(* IEC 61131-3 sources: Dev/Dev_V200/200 (part 11) *)

  	NH_M {HIDDEN} :  STRUCT 												 // m-stranka univerzalneho browsu
      // odtialto sa maze po prihlaseni
      naz         : STRING[20];                                // editovanie nazvu v hlavicke
      lvl         : USINT;                                     // level vnorenia
      lvp         : USINT;                                     // level + pg
      lng         : USINT;                                     // jazyk
      wht         : SINT;                                      // sposob ziskania dat do browsu
      iter        : SINT;                                      // iteracia
      delay       : UINT;                                      // cakanie medzi vykreslovanim (delay)
      new         : INT := -1;                                 // ND cislo pridaneho/najdeneho/vymazaneho riadka v ramci aCfg[cf]
      set         : BOOL;                                      // povolenie setup modu
      edt         : BOOL;                                      // prebieha editacia nazvu (tit)
      rgb         : BOOL;                                      // farba preRGB sa vybera aj cez slidery
      srt         : BOOL;                                      // moze preusporiadat riadky
      frm         : BOOL;                                      // aktivny vnoreny web iFrame (prekryje / deaktivuje can)
//      ref         : BOOL;                                      // prinak refreshu webu (ze prave bol refresh)
      htx         : USINT ;                                    // ktora webova stranka je zobrazena
      htt         : STRING; // := 'https://nachhouse.atlassian.net/secure/RapidBoard.jspa?rapidView=1&projectKey=NACH&selectedIssue=NACH-13' ;                             // webova adresa 'https:/www.nachhouse.sk'
      mno         : ARRAY[1..2] OF NH_OBJ_MNU;                 // zalohovanie horneho riadka pri editacii
      mnu         : ARRAY[0..3] OF NH_MNU;                    // menu
		lvd			: ARRAY[0..3] OF NH_LVL;						  // data jednotlivych vnoreni (level=lv)
      ixb         : ARRAY[0..1] OF NH_IXB;
      brw         : NH_BRW;                                   // brows
		pod			: NH_POD;
	END_STRUCT;

  	NH_WEB  {HIDDEN}:  STRUCT
		M			   : ARRAY[1.._Nh_WEB_M] OF NH_M;
      A           : ARRAY[1.._Nh_WEB_M] OF NH_CAN;
      nbr         : USINT;                         // ktory aWeb[nbr] je prave aktivny
      nrf         : USINT;								// actual count refresh display
      trg         : aTrg;
      Go          : BOOL;
	END_STRUCT;

  	NH_CAT_DSC {HIDDEN}:  STRUCT 					// categorie
 		Name        : STRING[13];
      typ         : SINT := 125;                   // filter CAT=recno(), alebo ak je > 99 tak zoznam
      dev         : USINT;                          // filter dev alebo ak je > 99 tak zoznam
      obr         : USINT := 12;
      ob0         : USINT;
      ob1         : USINT;
      Dsc         : STRING[25];

	END_STRUCT;

  	NH_STP_DSC {HIDDEN}:  STRUCT 					// categorie
 		Name        : STRING[13];
//      typ         : USINT := 255;                   // filter CAT=recno(), alebo ak je > 99 tak zoznam
      typ         : SINT := 125;                   // filter CAT=recno(), alebo ak je > 99 tak zoznam
      dev         : USINT;                          // filter dev alebo ak je > 99 tak zoznam
      obr         : USINT := 23;
	END_STRUCT;

END_TYPE

VAR_GLOBAL CONSTANT
   _e_NH_IDX_ROW        {HIDDEN}	   : NH_IDX_ROW;
	  eFilt_List			:  FILT_LIST;                                                                                      // prazdny filter
	  eFilt_List_typ		:  FILT_LIST_Typ;                                                                                      // prazdny filter

	  eRn     {HIDDEN} 	: NH_RUN_VAL2;

     eMnH     {HIDDEN} 	: NH_MNU := (     o := [(
                                        fn :=  1, wh :=  1, cm := 25  ), //       // logo
                                       (fn := 23, wh := 25, cm := 250  ),         // setup
                                       (fn :=  3, wh :=  0, cm := 20   ),         // home
                                       (fn := 41, wh := 42, cm := 21   ),         // FAV
                                       (fn := 16, wh := 17, cm := 22   ),         // rom
                                       (fn := 10, wh := 11, cm := 23   ),         // cat
                                       (fn := 27, wh := 28, cm := 24   ),         // act
                                       (fn := 49, wh :=  0, cm := 26   )]         // ON/OFF
                           );

      eMn0     {HIDDEN} : NH_MNU := (     o := [
                                       (fn :=  1, cm := 25),         // globalne nastaveia
                                       (fn := 23, cm := 250),        // setup ON/OFF
                                       (fn := 0),                    // home
                                       (fn := 41, cm :=  21),        // FAV
                                       (fn := 16, cm :=  22),        // rom
                                       (fn := 10, cm :=  23),        // cat
                                       (fn := 27, cm :=  24),        // act
                                       (fn := 0,)]);                 // ON/OFF

      eMn1     {HIDDEN} : NH_MNU := (     o := [(fn :=  0 ),  //  <
                                       (fn :=  0 ),  //  setup
                                       (fn :=  3,          cm :=  20),         // home
                                       (fn := 41,wh := 42, cm :=  21),         // FAV
                                       (fn := 16,wh := 17, cm :=  22),         // rom
                                       (fn := 10,wh := 11, cm :=  23),         // cat
                                       (fn := 27,wh := 28, cm :=  24),         // act
                                       (fn := 49,wh := 51, cm :=  26)]);       // ON/OFF

      eMvz      {HIDDEN} : NH_MNU := (     o := [(fn :=  6,wh :=   0,cm :=  31),       // <
                                       (fn :=   0,wh :=   6,cm :=   0, w:=72),  // obrazok vyssej casti
                                       (fn :=  35,wh :=  38,cm :=  33),          // 3 check
                                       (fn :=  10,wh :=  11,cm :=  34),          // 4 cat
                                       (fn :=  16,wh :=  18,cm :=  35),          // 5 all.rom / 1rom
                                       (fn := 348,wh := 348,cm :=  82),          // 6 priradit rom
//											      (fn :=  23,wh :=  24,cm :=  82),       	// 7-tune - parametre kurenia
//                                       (fn := 112,wh := 113,cm :=  36),          // visible
                                       (fn :=  39,wh :=  40,cm :=  37),          // 7-list     NESMIE SA OPRAVOVAT cm!!
                                       (fn :=  33,wh :=  34,cm :=  38)]);        // 8-play     NESMIE SA OPRAVOVAT cm!!

      eMn101     {HIDDEN} : NH_MNU := (   o := [(fn :=   6,wh :=   6,cm :=  31),          //  <
                                       (),
                                       (),
                                       (),
                                       (),
                                       (fn :=  23,wh :=  24,cm :=   3, x := xc)]);      // setup = Nastavenie parametrov

      eMn102     {HIDDEN} : NH_MNU := (   o := [(fn :=   6,wh :=   6,cm :=  31),          //  <
                                       (),
                                       (),
                                       (),
                                       (fn := 120,wh := 121,cm :=   1),          // Time
                                       (fn :=  23,wh :=  24,cm :=   3)]);        // setup = Nastavenie parametrov

      eMn103     {HIDDEN} : NH_MNU := (   o := [(fn :=   6,wh :=   6,cm :=  31),          //  <
                                       (),
                                       (fn := 122,wh := 123,cm :=   2,x:=xc-90),          // Level
                                       (fn :=  23,wh :=  24,cm :=   3,x:=xc   ),        // setup
                                       (fn :=  83,wh :=  84,cm := 121,x:=xc+90)]);           // tune predradnik / RGB

      eMn104     {HIDDEN} : NH_MNU := (   o := [(fn :=   6,wh :=   6,cm :=  31),          //  <
                                       (),
                                       (),
                                       (fn := 120,wh := 121,cm :=   1),             // Time
                                       (fn := 122,wh := 123,cm :=   2),             // Level
                                       (fn :=  23,wh :=  24,cm :=   3),             // setup
                                       (fn :=  83,wh :=  84,cm := 121)]);           // tune predradnik / RGB

      eMn105     {HIDDEN} : NH_MNU := (   o := [(fn :=   6,wh :=   6,cm :=  31),          //  <
                                       (),
                                       (fn := 120,wh := 121,cm :=   1,x:=xc-180),          // Time
                                       (fn := 122,wh := 123,cm :=   2,x := xc-90),          // Level + Ramp ON/OFF
                                       (fn := 124,wh := 125,cm :=   4,x := xc),          // COLOR
                                       (fn :=  23,wh :=  24,cm :=   3,x := xc+90),          // setup = Nastavenie parametrov
                                       (fn :=  83,wh :=  84,cm := 121,x := xc+180)]);        // tune predradnik / RGB

      eMnTLA   {HIDDEN} : NH_MNU := (   o := [(fn :=   6,wh :=   6,cm :=  31),          //  <
                                       (),
                                       (fn :=  33,wh :=  34,cm :=   5,x := 205),          // PLAY = priradenie
                                       (fn :=  23,wh :=  24,cm :=   6,x := 385)]);        // setup

      eMnWSB   {HIDDEN} : NH_MNU := (   o := [(fn :=   6,wh :=   6,cm :=  31),          //  <
                                       (),
                                       (fn :=  33,wh :=  34,cm :=   5,x := 205),          // PLAY = priradenie
                                       (fn := 204,wh := 205,cm := 120,x := 295),          // LED WSB
                                       (fn :=  23,wh :=  24,cm :=   6,x := 385)]);        // setup

      eMnPIR     {HIDDEN} : NH_MNU := (   o := [(fn :=   6,wh :=   6,cm :=  31),          //  <
                                       (fn :=   0,wh :=   0,cm :=   0),
                                       (fn :=   0,wh :=   0,cm :=   0),
                                       (fn := 215,wh := 216,cm :=  10,x := 115),          // Day
                                       (fn := 217,wh := 218,cm :=  10,x := 205),          // Evening
                                       (fn := 219,wh := 220,cm :=  10,x := 295),          // Night
                                       (fn := 221,wh := 222,cm :=  10,x := 385),          // Morning
                                       (fn :=  23,wh :=  24,cm :=   9,x := 475)]);        // setup = Nastavenie parametrov

      eMnUsr     {HIDDEN} : NH_MNU := (   o :=
                                      [(fn :=   6,wh :=   6,cm :=  31),          //  <
                                       (fn :=  32,wh :=  25,cm := 101),          //  +
                                       (fn :=   0,wh :=   0,cm :=   0),
                                       (fn :=   0,wh :=   0,cm :=   0),
                                       (fn :=  79,wh :=  79,cm :=  55),          // Users
                                       (fn := 285,wh := 286,cm :=  56),          // Web
                                       (fn :=   0,wh :=   0,cm :=   0),
                                       (fn :=   0,wh :=   0,cm :=   0)]);

(*
   _NhObrXYZ {HIDDEN} :  ARRAY [-10..-1,0..3] OF INT :=                 // obrazky podla nejakej podmieny (typ,stav...)
            [
//                21, 79,315, 21,             // -11 ZONE
               258, 82,  0,  0,             // -10 RH,CO2,CO
               508,216,166,507,             // -9 BRA  garaz,brana,branicka,zavora
               168,169,169,168,             // -8 SIR/STROB/
               183,184,185,186,             // -7 HET
                60, 60, 60, 60,             // -6  FAV dash/quick/FAV all/FAV user
                17, 19, 15,17,              // -5  ROM   In/OUT/pivnica
               106,107,  0,  0,             // -4  TLA   1/2
               102,103,104,105,             // -3  WSB   2/4/8/5
               100, 99,100,100,             // -2  termoventil : TVE, spirala
               161,162,  0,  0              // -1  teploty  :    miestnost,vonku //,podlaha,kotol

            ];

   // wht   :  index _NhStavDev[wht] odkial sa zoberi parametre do prikazu pre zobrazenie
   //          _NhVal2(wh := _NhStaDev[s].wht, obr := _NhStaDev[s].val);
   //             wh    - je bud podklad, alebo jednorazova prikaz, ktory nadefinuje vykreslenie
   //             obr   - ak si ho funkcia (wh) inak nespracuje, tak je to obrazok
   // val   :  ak je > 0 = cislo obrazka
   //          ak je < 0 je to odkaz na _NhObrXYZ[val], kde su obrazky podla nejakeho kriteria k DEV (vacsinou xCfg^.typ). rozduje funkcia _NhObrNbr()

   _NhObrDev  :  ARRAY [0.._Nh_CFG] OF NH_DEF_OBR :=     // definicia zakladnych obrazkov a obrazkov stavu (stav=odkaz) pre  DEV
            [
            (wht :=   0, val :=  23),      //  wht = index _NhStavDev[wht], val = cislo obrazka   ak je val < 0 potom je odkaz na _NhObrXYZ[val]
            (wht :=   1, val :=  -5),      //  1 ROM INR/EXT
            (wht :=   0, val :=  11),      //  2 CAT
            (wht :=   0, val :=  21),      //  3 ZON  stavovy obrazok sa definuje v _NhBrw6 CASE:9, hlavny obrazok:=21
            (wht :=  27, val :=  30),      //  4 SCN
            (wht :=  25, val :=  28),      //  5 ACT  0/34

//            (wht :=  29, val :=  -7),      //  6 HET
            (wht :=   0, val := 183),      //  6 HET
            (wht :=  42, val :=  95),      //  7 KOT
            (wht :=  42, val := 100),      //  8 TVE
            (wht :=   0, val := 101),      //  9 CER

            (wht :=   5, val :=  62),      // 10 SVD
            (wht :=   7, val :=  63),      // 11 SVA
            (wht :=   9, val :=  64),      // 12 RGB

            (wht :=   0, val :=  -3),      // 13 WSB     stavovy obrazok sa definuje v _NhBrw6
            (wht :=   0, val :=  -4),      // 14 TLA     stavovy obrazok sa definuje v _NhBrw6
            (wht :=  23, val :=  87),      // 15 PIR
            (wht :=   3, val :=  -1),      // 16 TER
            (wht :=   3, val := 163),      // 17 TEH
            (wht :=   3, val := 164),      // 18 TEK
            (wht :=   4, val :=  86),      // 19 LUX
            (wht :=   0, val :=  -6),      // 20 FAV
            (wht :=  11, val :=  73),      // 21 ZAS
            (wht :=   0, val :=  78),      // 22 USR
            (wht :=  30, val :=  70),      // 23 VENT
            (wht :=   0, val :=  97),      // 24 KEY
            (wht :=   0, val := 298),      // 25 SMART-WAY
            (wht :=   0, val :=   1),      // 26   POI
            (wht :=   0, val :=   1),      // 27 H2O
            (wht :=   0, val :=   1),      // 28 FIR
            (wht :=   0, val :=   1),      // 29 GAS
            (wht :=   0, val := 110),      // 30 MAR
            (wht :=  44, val := 114),      // 31 ROL
            (wht :=  30, val :=  -8),      // 32 SIR
            (wht :=  35, val :=  91),      // 33 DOR
            (wht :=  33, val :=  92),      // 34 WIN
            (wht :=   0, val := 197),      // 35 BLI
            (wht :=   0, val :=   1),      // 36   XXX
            (wht :=  50, val :=  -9),      // 37 BRA
            (wht :=   0, val :=   1),      // 38 RFI-snimace
            (wht :=   0, val :=   1),      // 39 RFK-karty
            (wht :=   0, val := 310),      // 40 TGL
            (wht :=   0, val := -10),      // 41 COX  (RH,CO2,CO)
            (wht :=   0, val := 290),      // 42 DALI-M
            (wht :=   0, val := 063),      // 43 DALI-S
            (wht :=   0, val := 029)       // 44 DALI-G
            ];

   // _NhStaDev: vykreslenie obraka podlastavu DEV vo funkcii : _NhVal2(wh := _NhStaDev[].wht, obr := _NhStaDev[].val);
   // jedno dev v _NhStaDev ma viac viet, podla stavu
   //    _NhStaDev[wht+0]  := 1.veta ked xDev^.ou.val = 0.0;
   //    _NhStaDev[wht+1]  := 2.veta ked xDev^.ou.val > 0.0;
   //    _NhStaDev[wht+2]  := 3.veta ked moze existovat ine kriterium unikatne k DEV

   // vsetko sa vyrobi v _NhShwObj() ked xO^.wh := 3

   _NhStaDev {HIDDEN} :  ARRAY [0.._Nh_CFG] OF NH_DEF_OBR :=               // zobrazenie stavy DEV (obrazky, hodnoty, ikony ,,,)
            [
            (wht :=   0, val :=  23),      //  0 nic (obrazok setup)
            (wht :=   1, val :=   0),        //  1 ROM - zobrazenie teploty
            (),                              // 2 - volne
//            (wht :=  18, val :=  66),        //  2 ZON - zobrazenie teploty
            (wht :=   1, val :=   0),        //  3 teplota miestnosti,vonku,podlahy,kotla... podla typ
            (wht :=   2, val :=   0),        //  4 LUX - zobrazenie osvetlenia
            (wht :=  10, val :=  -1),        //  5 SVD - OFF   (-1 znamena ze sa nevykresli ziadny obrazok !!!)
//            (wht :=  11, val :=   0),        //  6 SVD - ON - v zltom kruhu s gradientom
            (wht :=  17, val := 201),        //  6 SVD - ON - v zltom kruhu s gradientom
            (wht :=  10, val :=  -1),        //  7 SVA - OFF
//            (wht :=  12, val :=   0),        //  8 SVA - lvl v zltom kruhu s gradientom
            (wht :=  17, val := 201),        //  8 SVA - ON - v zltom kruhu s gradientom
            (wht :=  10, val :=  -1),        //  9 RGB - OFF
//            (wht :=  12, val :=   0),        // 10 RGB - lvl v zltom kruhu s gradientom
            (wht :=  17, val := 201),        // 10 RGB - ON - v zltom kruhu s gradientom

            (wht :=  18, val :=  73),       // 11 ZAS - NEURCENY-OFF            sivy + obrazok
            (wht :=  18, val :=  62),       // 12 ZAS - SVE-OFF                 sivy + obrazok
            (wht :=  18, val :=  50),       // 13 ZAS - STYKAC-OFF               sivy + obrazok
            (wht :=  18, val :=  61),       // 14 ZAS - HET-OFF                 sivy + obrazok
            (wht :=  18, val := 159),       // 15 ZAS - NABIJ.STANICA-OFF        sivy + obrazok
            (wht :=  18, val :=  73),       // 16 ZAS - rezerva-OFF              sivy + obrazok

            (wht :=  13, val := 202),       // 17 ZAS - NEURCENY-ON             zeleny + obrazok
            (wht :=  17, val := 201),       // 18 ZAS - SVD-ON                  zlty   + obrazok
            (wht :=  13, val := 213),       // 19 ZAS - SYKAC ON                 zeleny + obrazok
            (wht :=  13, val := 203),       // 20 ZAS - HET-ON                  zeleny + obrazok
            (wht :=  13, val := 214),       // 21 ZAS - NABIJACIA STANICA-ON    zeleny + obrazok
            (wht :=  13, val := 202),       // 22 ZAS - rezerva -ON             zeleny + obrazok

            (wht :=  10, val :=  -1),       // 23 PIR - pir je v klude, neodpocitava sa nic
            (wht :=  16, val :=  89),       // 24 PIR - prihadza signal          cierna postava v modrom

            (wht :=  18, val :=  28),       // 25 ACT - OFF sipka v sivom kruhu
            (wht :=  20, val :=  28),       // 26 ACT - ON sipka v Azurovom kruhu bez gradientu

            (wht :=  18, val :=  30),       // 27 SCN - OFF scn v sivom kruhu
            (wht :=  14, val := 207),       // 28 SCN - ON  scn v oranzovom kruhu

            (wht :=   1, val :=   0),       // 29 HET - zobrazenie teploty

            (wht :=  10, val :=  -1),       // 30 VEN - OFF
            (wht :=  13, val := 215),       // 31 VEN - ON - v modrom kruhu s gradientom

            (wht :=   4, val :=   0),       // 32 TVE - vystredene cislo v azurovom kruhu

            (wht :=  18, val :=  -1),       // 33 WIN - OFF
            (wht :=  14, val :=  92),       // 34 WIN - ON - v modrom kruhu s gradientom

            (wht :=  18, val :=  -1),       // 35 DOR - OFF
            (wht :=  14, val :=  91),       // 36 DOR - ON - v modrom kruhu s gradientom

            (wht :=  18, val :=  66),       // 37 ZON - Unlocked 0
            (wht :=  14, val :=  67),       // 38 ZON - Lock   1/2
            (wht :=  15, val :=  67),       // 39 ZON - Lock full
            (wht :=  18, val :=  66),       // 40 ZON - Locking
            (wht :=  18, val :=  66),       // 41 ZON - Unlocking

            (wht :=  10, val :=  -1),       // 42 TVE - OFF
            (wht :=  40, val :=   0),       // 43 TVE - cerveny kruh s cislo v strede

            (wht :=  18, val := 114),       // 44 ROL - OFF  0%      dn - zatiahnute     sivy
            (wht :=  14, val := 115),       // 45 ROL - viac 1-99%   up/dn - povytiahnute      oranzovy
            (wht :=  23, val := 117),       // 46 ROL - pohyb hore               cerveny
            (wht :=  23, val := 118),       // 47 ROL - pohyb dolu               cerveny
            (wht :=  90, val := 501),       // 48 ŽAL - zatienene    siva
            (wht :=  90, val := 500),       // 49 ŽAL - zodtienene   biela

            (wht :=  18, val := 509),       // 50 GAR - OFF  0%         sivy
            (wht :=  23, val := 510),       // 52 GAR - otvorene  100%  cerveny
            (wht :=  18, val := 216),       // 53 BRANA - OFF  0%         sivy
            (wht :=  15, val := 217),       // 54 BRANA - otvorene  100%  cerveny gradient
            (wht :=  18, val := 166),       // 55 BRANICKA - OFF  0%         sivy
            (wht :=  23, val := 167),       // 56 BRANICKA - otvorene  100%  cerveny
            (wht :=  21, val := 506),       // 55 BRANICKA - OFF  0%         sivy
            (wht :=  23, val := 507)        // 56 BRANICKA - otvorene  100%  cerveny

         ];

   // tito parametre sa posielaju do _NhVal2(wh := _NhStaCat[s].wht, obr := _NhStaCat[s].val);
   // wht : funkcia
   // val : obrazok
   // vsetko sa vyrobi v _NhShwObj() ked xO^.wh := 2
*)

END_VAR

VAR_GLOBAL CONSTANT

	{ $ IF _nh_Cust = 0 OR _Nh_CUST = 1} 	 // vsetko

      _ePg0   : NH_PG_HOME :=
      (
      Hom := ( ob := [
               ( wh:= 1, x := xc,     y := yyc- 30,  w := 180,  fn := 255 ),                                  // domcek
               ( wh:= 1, x := xc,     y := yyc- 55,  w :=  32,  fn := 0 ),                                   // day/night vnutri
               ( wh:= 0, x := xc+ 40, y := yyc-120,  w :=  32,  fn := 140 ),                                  // day/night vonku
               ( wh:= 1, x := xc,     y := yyc-  5,  w :=  80,  fn :=  92,   cm := 50,    cf := (c:=2, n:=17)),   // okno
               (),
//               ( x := xc+ 30, y := yc+ 90,  w :=  50,  wh := 0,  fn :=  92, h := -70, FgC := 1, BgC := 8,   cf := (c:=2, n:=18)),   // otvorene dvere ( h > 0 : vymaze aj kruh pod obrazkom)
               ( x := xc- 30, y := yyc+ 90,  w :=  50,  wh := 0,  fn := 111, h := -70, FgC := 8, BgC := 1,   cf := (c:=2, n:=23)),   // otvoreny garaz
               ( x := xc+100, y := yyc+ 20,  w :=  50,  wh := 0,  fn :=  77, h :=   0,                       cf := (c:=2, n:=24)),  // otvorena brana/branicka
               ( x := xc- 45, y := yyc-130,  w :=  75,  wh := 1,  fn := 132, h :=   0,                       cf := (c:=2, n:=11)),  // fotovoltaika

               ( wh:=4, x := xc-60, y := yyc+45, w:=58, h:=48, fn := 0, FgC := 0, BgC := 0,   cf := (c:=1, n:=1)),   // otvorene dvere ( h > 0 : vymaze aj kruh pod obrazkom)
               ( wh:=4, x := xc-60, y := yyc+45, w:=58, h:=48, fn := 91, cm := 50,   cf := (c:=2, n:=18)),   // otvorene dvere ( h > 0 : vymaze aj kruh pod obrazkom)
               (BgC := 13)
                     ]),

      dsh :=  ( ob := [

               (x := 0,      y:= 0, wh := 0),
               (x := xc,     y:= yyc-253, w := 130, wh := 2, cm:=50),   // 1.kruznica pod obr.1 prvy hore
               (x := xc+158, y:= yyc-183, w := 130, wh := 2, cm:=50),   // 2.kruznica pod obr.2
               (x := xc+210, y:= yyc- 25, w := 130, wh := 2, cm:=50),   // kruznica pod obr.3 - vprav v strede
               (x := xc+158, y:= yyc+133, w := 130, wh := 2, cm:=50),   // kruznica pod obr.4
               (x := xc,     y:= yyc+203, w := 130, wh := 2, cm:=50),   // kruznica pod obr.5 - dolu
               (x := xc-158, y:= yyc+133, w := 130, wh := 2, cm:=50),   // kruznica pod obr.6
               (x := xc-210, y:= yyc- 25, w := 130, wh := 2, cm:=50),   // kruznica pod obr.7 - vlavo v strede
               (x := xc-158, y:= yyc-183, w := 130, wh := 2, cm:=50)    // kruznica pod obr.8
                     ]),

      Qck :=  ( ob := [

               (x := xc-220, y := yy2-70, w := 64, wh := 0),                      // 1 - preve zprava
               (x := xc-220, y := yy2-65, w := 64, wh := 2, cm:=50),                      // 1 - preve zprava
               (x := xc-130, y := yy2-65, w := 64, wh := 2, cm:=50),
               (x := xc- 40, y := yy2-65, w := 64, wh := 2, cm:=50),
               (x := xc+ 50, y := yy2-65, w := 64, wh := 2, cm:=50),
               (x := xc+140, y := yy2-65, w := 64, wh := 2, cm:=50),
               (x := xc+230, y := yy2-65, w := 64, wh := 2, cm:=50),                      // 6 - posledne zlava
               (x := xc+320, y := yy2-65, w := 64, wh := 2, cm:=50),                      // 7 - dalej
               ()
                     ]),
      xy := [
               (),
               (x := 380, y := 275),
               (x := 490, y := 400),
               (x := 490, y := 562),
               (x := 380, y := 693),
               (x := 205, y := 693),
               (x :=  87, y := 569),
               (x :=  87, y := 400),
               (x := 200, y := 275)
               ],

      );

	{ $ END_IF }

	{ $ IF _Nh_CUST = 2} 	                // Futbal.stadion HE
      _ePg0 : NH_PG_HOME :=
      (
      Home := ( ob := [
               ( x := xc,    y:= yc- 20, w:= 600, wh:=1,          fn := 300 ),                    // futb.stadion
//               ( x := xc+15, y:= yc- 20, w:= 160, wh:=1,          fn := 301 ),                    // futb.stadion
               ()
                     ]),
      Dash :=  ( ob := [
               (x := xc-200, y:= yc+220, w := 110, wh := 2 , cf := (c := 2)),   // kruznica pod obr.1 prvy hore
               (x := xc-200, y:= yc+ 65, w := 110, wh := 2 , cf := (c := 2)),   // kruznica pod obr.2
               (x := xc-200, y:= yc-105, w := 110, wh := 2 , cf := (c := 2)),   // kruznica pod obr.3 - vprav v strede
               (x := xc-200, y:= yc-260, w := 110, wh := 2 , cf := (c := 2)),   // kruznica pod obr.4
               (x := xc+195, y:= yc-260, w := 110, wh := 2 , cf := (c := 2)),   // kruznica pod obr.5 - dolu
               (x := xc+195, y:= yc-105, w := 110, wh := 2 , cf := (c := 2)),   // kruznica pod obr.6
               (x := xc+195, y:= yc+ 65, w := 110, wh := 2 , cf := (c := 2)),   // kruznica pod obr.7 - vlavo v strede
               (x := xc+195, y:= yc+220, w := 110, wh := 2 , cf := (c := 2))    // kruznica pod obr.8
                     ]),

      Quick :=  ( ob := [

               (x := xc+320, y := y2-60, w := 64, wh := 2),
               (x := xc+230, y := y2-60, w := 64, wh := 2),
               (x := xc+140, y := y2-60, w := 64, wh := 2),
               (x := xc+ 50, y := y2-60, w := 64, wh := 2),
               (x := xc- 40, y := y2-60, w := 64, wh := 2),
               (x := xc-130, y := y2-60, w := 64, wh := 2),
               (x := xc-220, y := y2-60, w := 64, wh := 2),
               (x := xc-310, y := y2-60, w := 64, wh := 2),
               (),
               (w := 48, wh := 100)                    // weather
                     ]),

      );

      eMnHfs     : NH_MNU := (  n := 3,                                               // len obrazok HOME
                              o := [(fn :=  1),(fn := 0),
                                       (wh := 4, fn := 4, cm :=20, x:=xc, y:= y2+55),         // home
                                       (wh := 0, fn := 0, cm :=0 ),
                                       (wh := 0, fn := 0, cm :=0 ),
                                       (wh := 0, fn := 0, cm :=0 ),
                                       (wh := 0, fn := 0, cm :=0 ),
                                       (wh := 0, fn := 0, cm :=0 )
                                       ]);

   { $ END_IF }

	{ $ IF _Nh_CUST = 3} 	                // zimny stadion HE
      _ePgHome : NH_PG_HOME;
	{ $ END_IF }
END_VAR

//      pHet     : ARRAY[0..1,1..4] OF USINT := [170,172,174,176, 171,173,175,177];                                       // HeatMode */1/2/3/ manual/program
//      pTve     : ARRAY[0..1,0..3] OF USINT := [ 49,172,174,176,  52,173,175,177];                                       // Tve    Off/1/2/3/ manual/program

VAR_GLOBAL CONSTANT

(*
   // [OFF/ON, HET/TVE, A/1/2/3]      HET, TVE  OFF..ON    A,0,1,2,3              [0,OFF,            n] [0,ON,             n]
   _ObrHetPVP     {HIDDEN}   : ARRAY[ 0  ..  2, 0..   1,   0 ..    4] OF USINT := [222,170,172,174,176,  223,171,173,175,177, // HET: [0,OFF/ON, PRG/0/1/2/3/4 ]
                                                                                   222, 54,172,174,176,  223,193,173,175,177, // VEN: [1,OFF/ON, PRG/0/1/2/3/4 ]
                                                                                   220, 54,172,174,176,  221,193,173,175,177  // TVE: [2,OFF/ON, MAN/0/1/2/3/4 ]
*)

   _NhListObr     {HIDDEN}   : NH_LIST_OBR;
   _NhTypeMnu     {HIDDEN}   : NH_TYPE_MNU;
	_NhDsh			{HIDDEN}   : NH_DSH;
   _eRowHed       {HIDDEN}	  : NH_ROW_H;                   // cisla hlavicka riadka
   _eSld          {HIDDEN}	  : NH_SLD_DAT;
   _eFil          {HIDDEN}	  : NH_FIL;
   _eWht          {HIDDEN}   : NH_TCH_WHT;
   _eTch          {HIDDEN}	  : NH_TCH;                     // prazdny touch
   _eRowH         {HIDDEN}	  : NH_ROW_H;                    // prazdna hlavicka riadka
//   _ObjDay        {HIDDEN}   : NH_POI_DAY_XY;
   _NhObrLeds     {HIDDEN}   : ARRAY[1..4] OF USINT := [210,209,212,208];    // R,G,B,SH

//	_NhObjCfgBlk    :  NH_OBJ_DAT  :=          // PIR
//      (wh:= 0, x:=125,  y:=109,  w:=48, h:= 68, FgC:=4,  BgC:=2,  fn:=0            ); // 5 Blk
	_NhObjD1pir    :  NH_OBJ_DAT  :=          // PIR
      (wh:= 0, x:=125,  y:=109,  w:=50, h:=68 , FgC:=7,  BgC:=2,  fn:=0, cf:=(c:=5)); // 6 PIR day mde

END_VAR

VAR_GLOBAL
	aWeb			      : NH_WEB;

   yRn         {HIDDEN}     : NH_RUN_VAL2;

   xM          {HIDDEN}     : PTR_TO NH_M;
   xA          {HIDDEN}     : PTR_TO NH_CAN;
   xB          {HIDDEN}     : PTR_TO NH_BRW;
   xL		      {HIDDEN}     : PTR_TO NH_LVL;
   xF		      {HIDDEN}     : PTR_TO NH_FIL;
   xU          {HIDDEN}     : PTR_TO NH_MNU;
   xR          {HIDDEN}     : PTR_TO NH_ROW;
   xR2         {HIDDEN}     : PTR_TO NH_ROW;
   xRowO			{HIDDEN}     : PTR_TO NH_ROW_O;
	xS          {HIDDEN}     : PTR_TO NH_SLD_DAT;
   xO          {HIDDEN}     : PTR_TO NH_OBJ_DAT;
   xO2         {HIDDEN}     : PTR_TO NH_OBJ_DAT;
   xOh         {HIDDEN}     : PTR_TO NH_OBJ_123;
   xOh2        {HIDDEN}     : PTR_TO NH_OBJ_123;

   x4o         {HIDDEN}     : PTR_TO NH_OBJ_4O1;
	xRo 			{HIDDEN}		 : PTR_TO NH_OBJ_ROL;
//	yRo 			{HIDDEN}	AT aWeb.M[1].brw.r[14]	: NH_OBJ_ROL;
	yRo 			{HIDDEN}		:  NH_OBJ_ROL;
	x124			{HIDDEN}		:  PTR_TO NH_OBJ_124;
	y124			{HIDDEN}		:  NH_OBJ_124;

   xoDsh       {HIDDEN}     : PTR_TO NH_OBJ_DSH;

   xOm         {HIDDEN}     : PTR_TO NH_OBJ_MNU;
   xIxB        {HIDDEN}	    : PTR_TO NH_IXB;
   xIdx        {HIDDEN}	    : PTR_TO NH_IDX;
 	yIdxR			{HIDDEN}	    : NH_IDX_ROW;

   ky2          {HIDDEN} : INT := 915;                    // koniec browsu = zaciatok spodneho menu
   kyr          {HIDDEN} : INT := 132;                    // vyska riadku
   kyc          {HIDDEN} : INT := 510;                    // stred Y
   kyb          {HIDDEN} : INT := 800;                    // celkova vyska browsu
   yk           {HIDDEN}       : REAL;
   yLVL                   : NH_LVL;
   aAcc                             : NH_WEB_ACC;                      // riadiaca premenne
   CustomizedLoginPage AT %S355.1    {HIDDEN}   : BOOL := true;                     // povolenie Cust pristupu (prekopirovat XML do web/import)
   targetPage                        {HIDDEN} : STRING[20] := '001_NHM.XML';           // nazov stranky na ktoru presmeruje REDIR.XML
   aHtt                              {HIDDEN} : STRING[80] ; //:= '_NH_USR_.XML';
//   pageLogout                       : ARRAY [1..3] OF STRING[20];       //

END_VAR

VAR_GLOBAL		// docasne pomocne premenne
   yS          				{HIDDEN}     : NH_SLD_DAT;
   y4o         				{HIDDEN}     : NH_OBJ_4O1;
   yOh         				{HIDDEN}     : NH_OBJ_123;
	yoDsh       				{HIDDEN}     : NH_OBJ_DSH;
	_NhObjO4rom 				{HIDDEN}     :  NH_OBJ_4O1;
	_NhObjO4sta 				{HIDDEN}     :  NH_OBJ_4O2;
   xCan        				{HIDDEN}     : PTR_TO TCanvasData;
END_VAR

FUNCTION _NhVal2  : BOOL           // nadefinovanie stavoveho obrazka/textu pre kategoriu
   VAR_INPUT
      xy       : BOOL;                    // znamena, ze sa text vypisuje len pre to co je v x,y, inak pre xO^.x + x
      noxy     : BOOL;                    // text sa vypise od nastavenej pozicie
      nofmt    : BOOL;                    // text sa neformatuje
      crc      : BOOL;                    // vykresluje sa kruh
      box      : BOOL;                    // vykresluje sa obdlznik
      fil      : BOOL := true;            // vykresluje sa obsah kruhu/obdlznika
   	wrk		: BOOL;
	   wh       : USINT;                   // predvolba
      grd      : USINT;                   // typ gradientu
      obr      : INT;                     // vykresli sa obrazok
      txt      : SINT   := -1;            // vypise sa text (-1 := nic sa nevypise)
		nTxt		: INT;							// cislo textu
      FgC      : USINT  := 2;             // GCOLOR_LTGRAY;
      BgC      : USINT  := 1;             // GCOLOR_BLACK;
      FgT      : USINT  := 4;             // GCOLOR_WHILE;
      fmt      : INT    := 2;             // formatovanie textu (stred riadka, stred textu)
      wC       : INT    ;                 // priemer kruhu/sirka boxu
      hB       : INT    ;                 // vyska boxu
      wO       : INT    ;                 // velkost obrazka
      wT       : INT := 22   ;            // velkost textu
      wL       : USINT  := 2;             // hrubka kruznice / oramovanie kruhu
      x,y      : INT;                     // korekcie
      r        : INT    := 2;             // polomer Rounbow
      ob       : SINT := -1;               // namapuje xO
      val      : STRING[10];              // nieco naforpatovane pre zobrazenie ako text
   END_VAR
   VAR_TEMP
      n        : INT;
   END_VAR
   _NhVal2 := true;
   IF ob > -1 THEN
      xO := ADR(xR^.o.ob[ ob ]);
   END_IF;

   IF wC = 0 THEN
      wC := xO^.w;
   END_IF;
   IF wO = 0 THEN
//      wO := wC-7;
      wO := wC/5*4;
   END_IF;
   IF hB = 0 THEN
      hB := wC;
   END_IF;
   IF wT = 0 THEN
      wT := xO^.h;
   END_IF;
   CASE wh OF                                                          // jednoucelovo nadefinovane predvolby

      0: //bez predvolby = vypisuje sa podla toho co prislo v parametroch ( crc,obr,txt....)
         ;

    100: // normalna teplota z al.ou.val, formatovanie textu podla xO^.fn    , vyska xO^.h, farba podla FgC
         FgT := xO^.FgC; txt := 10; wT := xO^.h; fmt := xO^.fn; fil := false;
    101: // % (luxy,CO) z al.ou.val, formatovanie textu podla xO^.fn, vyska xO^.h
         FgT := xO^.FgC; txt := 11; wT := xO^.h; fmt := xO^.fn; fil := false;
    102: // oranzovy gradient-kruh s ciernym 'ON'
         fil :=1; crc := 1; grd := 11;  FgC :=15; BgC :=  4; FgT := 1; txt := 2; wT := 18;
    103: // azurovy gradient-kruh s ciernym 'ON'
         fil :=1; crc := 1; grd := 11;  FgC :=3; BgC :=  4; FgT := 1; txt := 2; wT := 18;

    109: // modry gradient-kruh s cislom v strede z al.ou.val
         fil :=1; crc := 1; grd := 11;  FgC := 3; BgC :=  3; FgT := 4; txt :=15; wT := 22; fmt := 2;
    110: // zlty gradient-kruh s cislom v strede z al.ou.val
         fil :=1; crc := 1; grd := 11;  FgC := 5; BgC :=  4; FgT := 1; txt :=15; wT := 22; fmt := 2;
    111: // Zeleny gradient-kruh s cislom v strede z al.ou.val
         fil :=1; crc := 1; grd := 11;  FgC := 8; BgC :=  4; FgT := 1; txt :=15; wT := 22; fmt := 2;
    112: // Oranzovy gradient-kruh s cislom v strede z al.ou.val
         fil :=1; crc := 1; grd := 11;  FgC :=15; BgC :=  4; FgT := 1; txt :=15; wT := 22; fmt := 2;
    113: // Azurovy  gradient-kruh s cislom v strede z al.ou.val
         fil :=1; crc := 1; grd := 11;  FgC := 3; BgC :=  4; FgT := 1; txt :=15; wT := 22; fmt := 2;
    114: // Purpurovy gradient-kruh s cislom v strede z al.ou.val
         fil :=1; crc := 1; grd := 11;  FgC := 28; BgC := 2; FgT := 4; txt :=15; wT := 22; fmt := 2;
    115: // Cerveny gradient-kruh s cislom v strede z al.ou.val
         fil :=1; crc := 1; grd := 11;  FgC := 7; BgC :=  4; FgT := 1; txt :=15; wT := 22; fmt := 2;
    116: // Biely gradient-kruh s cislom v strede z al.ou.val
         fil :=1; crc := 1; grd := 11;  FgC := 4; BgC :=  2; FgT := 1; txt :=15; wT := 22; fmt := 2;
    117: // Zeleny kruh bez grd s cislom z VR cierny text - pre CHECK/analog
	      fil :=1; crc := 1; grd := 1;  FgC := 8; BgC :=  8; FgT := 1; txt := 3; wT := 22; fmt := 2;
    118: // Zeleny kruh bez grd s cislom z VR cierny text - pre CHECK/DIGITAL
	      fil :=1; crc := 1; grd := 1;  FgC := 8; BgC :=  8; FgT := 1; txt := 2; wT := 22; fmt := 2;
    120: // silne sve tlo-cerveny  kruh + gradient
         fil :=1; crc := 1; grd := 11;  FgC := 18; BgC :=  4;   //BgC :=  4;

    150: // Cerveny gradient-kruh s cislom v strede z al.ou.sta
         fil :=1; crc := 1; grd := 11;  FgC := 7; BgC :=  4; FgT := 1; txt :=16; wT := 22; fmt := 2;
    151: // Cerveny gradient-kruh s cislom v strede z al.ou.ex
         fil :=1; crc := 1; grd := 11;  FgC := 7; BgC :=  4; FgT := 1; txt :=17; wT := 22; fmt := 2;

    160: // tmavo-cerveny kruh + svetly gradient
         fil :=1; crc := 1; grd := 11;  FgC :=28; BgC :=  4;
    161: // purpurovy kruh + tmavy gradient
         fil :=1; crc := 1; grd := 13;  FgC :=28; BgC :=  1;   //BgC :=  4;

    170: // tmavo-modry obdlznik bez gradientu
         fil :=1; box := 1; grd := 1;   FgC :=4; BgC :=  9;
    171: // svetlo-modry obdlznik bez gradientu
         fil :=1; box := 1; grd := 11;  FgC :=4; BgC := 22;   //BgC :=  4;

      1: // teplota v browse
         FgT := xO^.FgC; txt := 10; wT := 32; fmt := 1; x := 30; y := -5;    // skoriguje suradnice vypisu teploty - posunie do prava a odtial sa vykresluje do lava
//         FgT := xO^.FgC; txt := 10; wT := xO^.h; fmt := 1; x := 30; y := -5;    // skoriguje suradnice vypisu teploty - posunie do prava a odtial sa vykresluje do lava
      2: // % osvetlenia v browse
         FgT := xO^.FgC; txt := 11; wT := 28; fmt := 1; x := 30; y := -5;
      3: // lx v browse
         FgT := xO^.FgC; txt := 12; wT := 28; fmt := 1; x := 30; y := -5;
      4: // vystredene cislo v sivom kruhu s gradientom
         FgT := 4; txt := 3; wT := 20; fmt := 2;               // cislo bielou
         crc := 1; grd := 11;  FgC := 2; BgC :=  1; wC := 60;

      9: // kruh bez gradientu vypln farbou Bgc, bez oramovanie pripadny text farbou FgC, text podla poslanych parametrov
         fil :=1; crc := 1; grd := 2; Fgc:= BgC; FgT := 1; wL := 0;

//         fil :=1; crc := 1; grd := 2;  FgC := 8; BgC :=  8; FgT := 1;

     10: // sivy gradient-kruh s bielym 'OFF'
         fil :=1; crc := 1; grd := 11;  FgC := 2; BgC :=  1; FgT := 4; txt := 1; wT := 19;

     11: // zlty gradient-kruh s ciernym 'ON'
         fil :=1; crc := 1; grd := 11;  FgC := 5; BgC :=  4; FgT := 1; txt := 2; wT := 18;

     12: // zlty gradient-kruh s cislom v strede
         fil :=1; crc := 1; grd := 11;  FgC := 5; BgC :=  4; FgT := 1; txt := 3; wT := 22;

     13: // zeleny   kruh + gradient
         fil :=1; crc := 1; grd := 11;  FgC := 8; BgC :=  4;
     14: // oranzovy kruh + gradient
         fil :=1; crc := 1; grd := 11; FgC := 15; BgC :=  4; //FgC := 6; BgC :=  4;
         IF obr > 0 THEN
            wO := wC/4*3;
         END_IF;
     15: // sve tlo-cerveny  kruh + gradient
         fil :=1; crc := 1; grd := 11;  FgC := 7; BgC :=  4;   //BgC :=  4;
     16: // azurovy  kruh + gradient
         fil :=1; crc := 1; grd := 11;  FgC := 3; BgC :=  4;
     17: // zlty gradient-kruh
         fil :=1; crc := 1; grd := 11;  FgC := 5; BgC :=  4;
     18: // sivy gradient-kruh
         fil :=1; crc := 1; grd := 11;  FgC := 2; BgC :=  1;
     19: // oranzovy kruh + gradient v strede oranzova, dooloko biela
         fil :=1; crc := 1; grd := 12;  FgC := 6; BgC := 26;
//         crc := 1; grd := 11;  FgC := 6; BgC := 4;

     20: // azurovy kruh bez gradientu
         fil :=1; crc := 1; grd := 2;  FgC := 3; BgC := 3; FgT := 4;
     21: // zelena  bez gradienu
         fil :=1; crc := 1; grd := 2;  FgC := 8; BgC :=  8; FgT := 1;
     22: // oranzova  bez gradientu
         fil :=1; crc := 1; grd := 2;  FgC := 6; BgC :=  6; FgT := 1;
     23: // cervena  bez gradientu
         fil :=1; crc := 1; grd := 2;  FgC := 7; BgC :=  7; FgT := 4;
     24: // biela  bez gradientu
         fil :=1; crc := 1; grd := 2;  FgC := 4; BgC :=  4; FgT := 1;

     25: // azurovy  bez gradient  + ON
         fil :=1; crc := 1; grd := 11;  FgC := 3; BgC :=  4; FgT := 1; txt := 2; wT := 24;
     26: // azurovy  kruh + \\gradient  + ON
         fil :=1; crc := 1; grd := 11;  FgC := 3; BgC :=  4; FgT := 1; txt := 2; wT := 24;

     27: // cierny kruh bez gradientu
         fil :=1; crc := 1; grd := 2;  FgC := 1; BgC := 1;

     28: // svetlo-purpurovy bez gradientu
//         fil :=1; crc := 1; grd := 2;  FgC := 28; BgC := 28;
         fil :=1; crc := 1; grd := 10;  FgC := 21; BgC :=21; FgT := 1; //txt := 0; wT := 44; fmt := 2;

     29: // zlty gradient-kruh s cislom v strede, vypisuje to co je xO^.fmt
         fil :=1; crc := 1; grd := 11;  FgC := 5; BgC :=  4; FgT := 1; wT := 22;

//     30: // sivy gradient-kruh s cislom v strede z yTx1
//         fil :=1; crc := 1; grd := 11;  FgC := 2; BgC :=  1; FgT := 4; txt := 0; wT := 44; fmt := 2;

     30: // tmavy modry gradient-kruh
//         fil :=1; crc := 1; grd := 11;  FgC := 9; BgC :=21; FgT := 1; //txt := 0; wT := 44; fmt := 2;
//         fil :=1; crc := 1; grd := 11;  FgC := 9; BgC :=1; FgT := 1; //txt := 0; wT := 44; fmt := 2;
//         fil :=1; crc := 1; grd := 11;  FgC :=20; BgC :=0; FgT := 4; //txt := 0; wT := 44; fmt := 2;
         fil :=1; crc := 1; grd := 11;  FgC :=3; BgC :=0; FgT := 4; //txt := 0; wT := 44; fmt := 2;

     31: // tmavy zeleny gradient-kruh
         fil :=1; crc := 1; grd := 11;  FgC := 8; BgC :=  1; //FgT := 4; txt := 0; wT := 44; fmt := 2;
     32: // tmavy oranzovy  gradient-kruh
         fil :=1; crc := 1; grd := 11;  FgC := 6; BgC :=  1; //FgT := 4; txt := 0; wT := 44; fmt := 2;
     33: // tmavy cerveny gradient-kruh
         fil :=1; crc := 1; grd := 10;  FgC := 1;  BgC :=  7; //FgT := 4; // txt :=9; wT := 38; fmt := 2;
     34: // tmavy azurovy gradient
         fil :=1; crc := 1; grd := 11;  FgC := 3;  BgC :=  1;// FgT := 4; txt := 0; wT := 44; fmt := 2;
     35: // biely gradient
         fil :=1; crc := 1; grd := 11;  FgC := 4; BgC :=  2; FgT := 1;
     36: // sivy  bez gradienu
         fil :=1; crc := 1; grd := 2;  FgC := 2; BgC :=  2; FgT := 1;
     37: // modry  bez gradienu
         fil :=1; crc := 1; grd := 2;  FgC := 9; BgC :=  9; FgT := 1;
     38: // tmavo-purpurovy bez gradientu
         fil :=1; crc := 1; grd :=12;  FgC := 1; BgC :=28;

     40: // cerveny bez gradient u kruh s cislom v strede
         fil :=1; crc := 1; grd := 2;  FgC := 7; BgC :=  7; FgT := 4; txt := 3; wT := 25;

     50: // sivy obdlznik
         fil :=1; crc := 0; box := 1; grd := 11;  FgC := 2; BgC :=  1;   wC := xO^.w; hB := xO^.h; wO := wC;

     52: // oranzovy obdlznik
         fil:=1; crc := 0; box := 1; grd := 11;  FgC := 6; BgC :=  4;   wC := xO^.w; hB := xO^.h; wO := wC;

     80: // podfarbenie menu
         fil :=1; crc := 0; box := 1; grd := 10;  FgC := 3; BgC := 27;   wC := xO^.w+10; hB := xO^.h+25;    //wO := wC;

     90: // bez podkladu, farba
         crc := 0; box := 0;
    ELSE // neurceny obr - svetlo-sivy grdirnt-kruh s obrazko setup
         crc := 1; grd := 11; FgC := 2; BgC :=  26; obr := 24;
   END_CASE;
   // vyberie gradient/frame

   IF grd > 0 THEN                                                         // ak je grd=0 akceptuju sa existujuce nastavenia
      CASE grd OF                                                          // kruznica, kruh, kruh s oramovanim, kruh s gradientom
          1 :  rmp := GFILL_STYLE_BGCOLOR;                                    // kruh bez oramovania bez gradientu
          2 :  rmp := GFILL_STYLE_FRAME;                                      // kruh s oramovanim bez gradientu
         10 :  rmp := GGRADIENT_STYLE_LINEAR;                                 // kruh s gradientom linear
         11 :  rmp := GGRADIENT_STYLE_LINEAR+GGRADIENT_STYLE_HORIZONTAL;      // kruh s gradientom linear+horizontal
         12 :  rmp := GGRADIENT_STYLE_RADIAL;                                 // kruh s gradientom RADIAL
         13 :  rmp := GGRADIENT_STYLE_RADIAL1_3;                            // kruh s gradientom RADIAL
         14 :  rmp := GGRADIENT_STYLE_BAR1_3;                            // kruh s gradientom RADIAL
      END_CASE;
      // nastavi gradient
      IF grd > 9 THEN                                                      // bude gradient
         GC_SetFillStyle      (style := GFILL_STYLE_GRADIENT, GrData := xCan);
         GC_SetGradientStyle  (style := rmp, color1 := _NhColor[FgC], color2 := _NhColor[BgC],  GrData := xCan);
      ELSE
         GC_SetFillStyle      (style := rmp, GrData := xCan);
         GC_SetLineWidth      (Width := wL,  GrData := xCan);
         IF FgC = 255 THEN
            GC_SetFgColor (Color 	:= _NhColor[0] ,GrData := xCan);		     // farba pozadia
            GC_SetBgColor (Color 	:= RGBA_TO_COLOR(r := rgb.R, g := rgb.G, b := rgb.B) ,GrData := xCan);		     // farba pozadia
         ELSE
            GC_SetFgColor (Color := _NhColor[FgC]    , GrData := xCan);
            GC_SetBgColor (Color := _NhColor[BgC]    , GrData := xCan);
         END_IF;
      END_IF;
   END_IF;
      IF noxy THEN
         ;
      ELSIF xy THEN
         GC_MoveTo   (x := x, y := y , GrData := xCan);
      ELSE
         GC_MoveTo   (x := xO^.x + x, y := xO^.y + y , GrData := xCan);
      END_IF;

   IF crc THEN
      GC_CCircle   (fill  := fil, r:= wC / 2,   GrData := xCan);  // kruznica                       2000:
   END_IF;
   IF box THEN
      GC_CRoundBox(fill  := fil, width := wC, height := hB,  r := r , GrData := xCan);
   END_IF;
   IF obr > 0 THEN
      GC_CImage   (filename := _NhFnObr(fn := obr), width := wO, height := wO,	GrData := xCan);
   END_IF;
	wrk	:= true;
   IF txt > -1 THEN
      CASE txt OF
        0 : ; // vypise sa to co je v yTx1
        1 : yTx1 := 'OFF';
        2 : yTx1 := 'ON';
        3 : yTx1 := USINT_TO_STRINGF(REAL_TO_USINT(vr),'%u');                      // vystredene cislo
        7 : yTx1 := REAL_TO_STRINGF(vr,'%7.1f°');                                  // vystredena teplota
            aTrim(txt := ADR(yTx1), wht := 3);
        8 : yTx1 := REAL_TO_STRINGF(vr,yTx2);                                      // hodnota naformatovana podla yTx2
//        10: yTx1 := REAL_TO_STRINGF(vr,'%7.1f°');                                  // teplota v browse
//        11: yTx1 := REAL_TO_STRINGF(vr,'%5.0f%%');                                 // % osvetlenia v browse
         9: yTx1 := REAL_TO_STRINGF(xDev^.al.ou.val,'%3.0f°');    						// teplota home
        10: yTx1 := REAL_TO_STRINGF(xDev^.al.ou.val,'%6.1f°');                                  // teplota v browse
            aTrim(txt := ADR(yTx1), wht := 3);
        11: yTx1 := REAL_TO_STRINGF(xDev^.al.ou.val,'%5.0f%%');                                 // % osvetlenia v browse
            aTrim(txt := ADR(yTx1), wht := 3);
        12: yTx1 := UINT_TO_STRINGF(xDev2^.al.et,'%d lx');                         // luxy ????
        13: yTx1 := 'GO';
        14: yTx1 := 'STOP';
//        15: yTx1 := REAL_TO_STRINGF(xDev^.al.ou.val,'%3.0f%');                                 // % osvetlenia v browse
        15: yTx1 := USINT_TO_STRINGF(REAL_TO_USINT(xDev^.al.ou.val),'%u');                  // cislo 0..255
        16: yTx1 := USINT_TO_STRINGF(xDev^.al.sta,'%u');
        17: yTx1 := INT_TO_STRINGF(xDev^.al.ex,'%u');
       100: yTx1 := yTx2;
       101: IF xO^.cf.c > 0 THEN
               _NhxPt(c := xO^.cf.c, n := xO^.cf.n, x:=7);                               // nazov DEV
               yTx1 := xPt^.cf.Name;
               yTx1 := LEFT(yTx1,xO^.w/8);
            ELSE
               yTx1 := '_NhVal2(txt=101)';
            END_IF;
            aTrim(txt := ADR(yTx1), wht := 3);
       102: yTx1  := xO^.fmt;
      END_CASE;
	ELSIF txt = -2 THEN
		IF nTxt > 0 THEN
		  _Nh_Lang(id := nTxt ,txt := ADR( yTx1 ));
		ELSE
			wrk := false;
		END_IF;
	ELSE
		wrk	:= false;
	END_IF;
	IF wrk THEN
	   IF nofmt THEN
         ;
      ELSIF fmt > 9 THEN                                                             // pod textom bude vymazany box farbou pozadnia
         vai := _Nh_Sty[fmt-10];  // + GTEXT_STYLE_FILLBG;
         GC_SetFillStyle   (style := GFILL_STYLE_BGCOLOR , GrData := xCan);
         GC_SetFgColor     (Color := _NhColor[0]    , GrData := xCan);          // farba ramceka
         GC_SetBgColor     (Color := _NhColor[0]    , GrData := xCan);          // farba podkladu
         GC_CBox           (fill  := fil, width := xO^.w+2 , height := wt + 4 ,   GrData := xCan);  // podklad pod textom
         GC_SetTextstyle(style   := vai               , GrData := xCan);           // formatovanie textu zlava do prava
      ELSIF fmt = -1 THEN                                                             // pod textom bude vymazany box farbou pozadnia
         GC_SetFillStyle(style   := GFILL_STYLE_BGCOLOR, GrData := xCan);
      ELSIF fmt = -2 THEN                                                             // pod textom bude vymazany box farbou pozadnia
         GC_SetTextstyle(style   := INT_TO_UINT(fmt)  , GrData := xCan);           // formatovanie zlava do prava
      ELSE
         vai := _Nh_Sty[fmt];                                                       // format textu bez podkladu
         GC_SetTextstyle(style   := vai               , GrData := xCan);           // formatovanie textu
      END_IF;
      GC_SetTextSize (size 	:= INT_TO_USINT(wt) , GrData := xCan);           // vyska textu
      GC_SetFgColor  (Color 	:= _NhColor[FgT]    , GrData := xCan);           // farba textu
      GC_WriteText   (text    := yTx1             , GrData := xCan);           //
   END_IF;
END_FUNCTION

FUNCTION _webState {HIDDEN} : USINT
   VAR_INPUT
      s     : T_SESSION_STATE;
   END_VAR
   CASE s OF
      SESSION_EMPTY     : _webState:=0; yTx3 := 'EMPTY  ';    // Spojení je volné
      SESSION_LOGIN     : _webState:=1; yTx3 := 'LOGIN.B';    // Zahájení prihlášení uživatele k web serveru
      SESSION_LOGIN_RUN : _webState:=2; yTx3 := 'LOGIN.R';    //Probíhá prihlašování uživatele k web serveru
      SESSION_ACTIVE    : _webState:=3; yTx3 := 'ACTIVE ';    //Probíhá komunikace s úspešne prihlášeným uživatelem
      SESSION_LOGOUT    : _webState:=4; yTx3 := 'LOGOUT ';    // Probíhá odlašování uživatele (ukoncuje se spojení)
      ELSE                _webState:=5; yTx3 := '???    ';
   END_CASE;
END_FUNCTION

FUNCTION _NhTchXY {HIDDEN} : BOOL    // dotyk nad bodom s rozptylom medzi hranicami  v1...v...v2
   VAR_INPUT
      v      : INT;
      v1     : INT;
      v2     : INT;
      xy     : INT := 20;
   END_VAR
   _NhTchXY := true;
   IF v >= v1 - xy  AND                                       // nie na hranica
      v <= v2 + xy THEN
      RETURN;
   END_IF;
   _NhTchXY := false;
END_FUNCTION

FUNCTION _NhShwMnu {HIDDEN}  : BOOL              // preberie ciastocne MENU z predchadzajucej urovne
   VAR_TEMP
      fn    : INT;
   END_VAR
      GC_SetFillStyle      (style := GFILL_STYLE_GRADIENT, GrData := xCan);
//      IF xL^.obj = 34 OR xL^.obj = 36 THEN     // IOV,FVL
      IF xL^.chk  THEN        // IOV,FVL
//         GC_SetGradientStyle  (style := GGRADIENT_STYLE_LINEAR, color1:= GCOLOR_BLACK, color2:=GCOLOR_GREEN+GCOLOR_TRANSPARENT1_4, GrData := xCan);
         GC_SetGradientStyle  (style := GGRADIENT_STYLE_LINEAR, color1:= GCOLOR_BLACK, color2:=GCOLOR_GREEN, GrData := xCan);
         GC_RoundBox          (fill:=1, r:=10, x:= 5, y:= 5, width := x2 ,height := y1-5, GrData := xCan);                    // horny modry podklad
      	GC_SetFgColor        (Color 	:= GCOLOR_WHITE, GrData := xCan);                                                         // nadpis cierna /zaelena
      ELSE
         GC_SetGradientStyle  (style := GGRADIENT_STYLE_LINEAR, color1:= GCOLOR_BLACK, color2:=GCOLOR_AZURE, GrData := xCan);
         GC_RoundBox          (fill:=1, r:=5, x:= 0, y:= 0, width := x2 ,height := 105, GrData := xCan);
      	GC_SetFgColor        (Color 	:= GCOLOR_WHITE, GrData := xCan);
      END_IF;
      // vymazat priestor spodneho menu
      GC_SetFillStyle      (style := GFILL_STYLE_BGCOLOR, GrData := xCan);
      GC_SetBgColor        (Color 	:= _NhColor[0] ,GrData := xCan);		                                                    // farba pozadia
      GC_Box               (fill:=1, x:= x0, y:= ky2, width := x2 ,height := 130, GrData := xCan);
      // obrazky
      FOR i := 1  TO 8 DO
         x := xU^.o[i].w;
         IF xU^.o[i].kxy = false THEN
            xU^.o[i].y  := REAL_TO_INT(INT_TO_REAL(xU^.o[i].y) * yk);
            xU^.o[i].kxy := true;
         END_IF;

         GC_MoveTo   (x :=xU^.o[i].x, y := xU^.o[i].y, GrData := xCan);
         IF i = xU^.n THEN       // podfarbenie vybrateho menu
            GC_SetFillStyle      (style := GFILL_STYLE_GRADIENT, GrData := xCan);
            IF xL^.chk THEN     // IOV,FVL
//               GC_SetGradientStyle  (style := GGRADIENT_STYLE_LINEAR, color2:= GCOLOR_BLACK, color1:=GCOLOR_GREEN+GCOLOR_TRANSPARENT1_4, GrData := xCan);
               GC_SetGradientStyle  (style := GGRADIENT_STYLE_LINEAR, color2:= GCOLOR_BLACK, color1:=GCOLOR_GREEN, GrData := xCan);
            ELSE
               GC_SetGradientStyle  (style := GGRADIENT_STYLE_LINEAR, color2:= GCOLOR_AZURE + GCOLOR_TRANSPARENT3_4 , color1:=GCOLOR_AZURE, GrData := xCan);
            END_IF;
            GC_CRoundBox          (fill:=1, r:=15, width := x ,height := x, GrData := xCan);
            fn := xU^.o[i].wh;                                                                                  // obrazok, ked je mnu vybrate
            x  := x - 5;
         ELSE
//            GC_MoveTo   (x :=xU^.o[i].x, y := xU^.o[i].y, GrData := xCan);
            fn := xU^.o[i].fn;                                                                                                // len zobrazit, nie vybrat
         END_IF;
         IF fn <> 0 THEN
            GC_CImage   (filename := _NhFnObr(fn := fn ), width := x, height := x,	GrData := xCan);
         END_IF;
      END_FOR;
      GC_SetFillStyle      (style := GFILL_STYLE_BGCOLOR, GrData := xCan);					                                        // farba neaktivnej ciary
     	GC_SetBgColor        (Color 	:= _RgbBck ,GrData := xCan);		                                                          // farba pozadia
      // text
      GC_MoveTo            (x := xc , y := xU^.o[1].y , GrData := xCan);
      GC_SetTextSize       (size 	:= 32, GrData := xCan);                            // vyska textu je aj pre hodnotu aj pripadny text
      GC_SetTextstyle      (style := _Nh_Sty[2], GrData := xCan);
		GC_CWriteText        (text := xL^.naz, GrData := xCan);
      // ciara
     	GC_SetFgColor        (Color 	:= GCOLOR_GRAY,GrData := xCan);		// farba aktivnej ciary
      GC_SetLineWidth      (Width := 2, GrData := xCan);
      GC_SetLineStyle      (style := GLINE_CAP_ROUND + GLINE_STYLE_SOLID, GrData := xCan);
      GC_Line              (y1 := ky2, y2 := ky2, x1:= 20, x2 := x2-20,GrData := xCan);
END_FUNCTION

FUNCTION _NhVazPar {HIDDEN} : BOOL  //
         IF xR^.h.in THEN
            xR^.h.cf       := xVaz^.in;                                    // preberie sa aj s parametrami
            xR^.o.ob[1].cf := xVaz^.in;
            xR^.o.ob[2].cf := xVaz^.in;
            xR^.o.ob[4].cf := xVaz^.ou;
         ELSE
            xR^.h.cf       := xVaz^.ou;
            xR^.o.ob[1].cf := xVaz^.ou;
            xR^.o.ob[2].cf := xVaz^.ou;
            xR^.o.ob[4].cf := xVaz^.in;
         END_IF;
END_FUNCTION

FUNCTION _NhUsrPar  {HIDDEN} : BOOL  // nastavi aktualne zobrazenie pre usra do menu[2], xL^.dsh
   VAR_INPUT
      sav      : BOOL;                 // true = ulozi k usrovi , false =  precita z usra
      fav      : BOOL;                 // favorite
      dsh      : BOOL;                 // dash
//      qck      : BOOL;
      ds1      : BOOL;
      qc1      : BOOL;
      usr      : USINT;                // ak je > 0 pouzije sa, inak aktualny user
   END_VAR
   _NhUsrPar   := true;
   IF usr = 0 THEN
      usr := xA^.usr;
   END_IF;
   _NhxPtU(c := 22, n :=usr ,x:=-1); xUsr := xPt;                                                // namapuje usra
   IF fav   THEN
      IF sav THEN
         xUsr^.cx.fav := xA^.fav;
      ELSE
         xA^.fav := xUsr^.cx.fav;
      END_IF;
   END_IF;
   IF ds1   THEN
      IF sav THEN
         xUsr^.cx.ds1 := xL^.rw1;
      ELSE
         xL^.rw1 := xUsr^.cx.ds1;
      END_IF;
   END_IF;
   IF qc1   THEN
      IF sav THEN
         xUsr^.cx.qc1 := xL^.rw1;
      ELSE
         xL^.rw1 := xUsr^.cx.qc1;
      END_IF;
   END_IF;
   IF dsh   THEN
      IF sav THEN
         xUsr^.cx.Brw[xL^.obj] := xL^.dsh;                  // ulozi cislo DSH k browsu
      ELSE
         xL^.dsh := xUsr^.cx.Brw[xL^.obj];
      END_IF;
   END_IF;
END_FUNCTION

FUNCTION  _Nh_Brw_Dsh_Chg   {HIDDEN}    : BOOL  // nastavi aktualne zobrazenie pre usra do menu[2], xL^.dsh
   VAR_INPUT
      chg      : BOOL;
      mnu      : USINT := 1;                                         // default je horne lave menu
   END_VAR
   _Nh_Brw_Dsh_Chg := true;
   xL^.dsh := LIMIT(1,xL^.dsh,4);										// opravi ak treba
   IF xA^.usr = 0 THEN														// ziadny user nastavi default
      _Nh_Brw_Dsh_Chg 		:= 0;
      xL^.dsh   				:= 1;                                                  // nacita aktualny dsh
      RETURN;
   END_IF;

	IF xUsr^.cx.DshSet THEN													// user moze menit
	   IF xL^.obj <= 30 THEN
   	   xL^.dsh := LIMIT(1,xUsr^.cx.brw[ xL^.obj ],3);  // nacita a nastavi ulozeny dsh
	   END_IF;
	   IF chg THEN                                              // pri zmene
   	   xL^.dsh := xL^.dsh + 1;
	   END_IF;
   	CASE xL^.dsh OF
	      2 :   ix 		:= 157;
   	   3 :   ix 		:= 158;
	   ELSE     ix 		:= 156;
   	         xL^.dsh 	:= 1;
	   END_CASE;
	   IF xL^.obj <= 30 THEN

//   	   _NhSysUpd(chg := xUsr^.cx.brw[ xL^.obj ] <> xL^.dsh);

      	xUsr^.cx.brw[ xL^.obj ] := xL^.dsh;                            // ulozi k usrovi
	   END_IF;
   	IF mnu > 0 THEN                               // rezim meny dsh
      	xU^.o[mnu].fn    := ix;                                        // prepnutie zobrazenie dash / riadok
	      xU^.o[mnu].cm    := 43;                                        // funkcia z menu
		ELSE
      	xU^.o[mnu].fn    := 0;                                        // prepnutie zobrazenie dash / riadok
	      xU^.o[mnu].cm    := 0;                                        // funkcia z menu
   	END_IF;
	   xL^.obd          := mnu;                                        	// funkcia z menu
	END_IF;
END_FUNCTION

FUNCTION _NhTchObjXYW {HIDDEN}: BOOL   // dotyk nad objektom X,Y,W
   VAR_INPUT
      x  :  INT;  // Lavy zaciatok objektu
      y  :  INT;  // nad objektom
      w  :  INT;  // sirka objeku
		h	:  INT := -1;	// vyska
   END_VAR
	IF h = -1 THEN
		h	:= w;
	END_IF;
   IF xA^.tch.x1 >= x 		AND                 // zaciatok X
      xA^.tch.x1 <= x + w 	AND                 // koniec X
      xA^.tch.y1 >= y  		AND                 // y-navrchu
      xA^.tch.y1 <= y + h  THEN                // y-spodok
      _NhTchObjXYW := true;
   ELSE
      _NhTchObjXYW := false;
   END_IF;
END_FUNCTION

VAR_GLOBAL
	yR 	: NH_ROW;
END_VAR

FUNCTION _Nh_Web_SHW_107 {HIDDEN} : BOOL      // vykreslit doplnujuce objektynad hlavnym objektom, dotyk a cykonanie pripadneho CMD
   VAR_INPUT
      tch      : BOOL;
 		row		: bool;
		obj		: SINT;
   END_VAR
   VAR
      x,y,o      : INT;
      r			: USINT;
   END_VAR
	yR		:= xR^;
   x4o   := xO;
   _Nh_Web_SHW_107 := false;
   FOR i := 1 TO 4 DO
      IF x4O^.ok[i] THEN
//y4O := x4O^;
			r := x4O^.obj;
			IF row THEN
				xO2 := ADR(xB^.r[ r ].o.ob[obj]);
			ELSE
				xO2 := ADR(xR^.o.ob[ r ]);
			END_IF;
   		grp   := xO2^.w * 10 / 28;                  // suradnica posunu vypocitana podla velkosti objektu
   	   x     := xO2^.x;
      	y     := xO2^.y;
         CASE i OF
            1: x  := x  - grp;
               y  := y  - grp;
            2: x  := x  + grp;
               y  := y  - grp;
            3: x  := x  - grp;
               y  := y  + grp;
            4: x  := x  + grp;
               y  := y  + grp;
         END_CASE;
         grp   := USINT_TO_INT(x4o^.wxy[i]);
         IF tch THEN
            IF _NhTchObjXYW(x:=x-grp/2, y:=y-grp/2, w:=grp) AND x4o^.cmd[i] > 0 THEN
               xA^.tch.cmd := x4o^.cmd[i];
               xA^.tch.cm  := x4o^.cmd[i];
//               xR^.o.ob[ x4O^.obj ].tch := false;
               _Nh_Web_SHW_107 := true;
               EXIT;
            END_IF;
//            xO^.tch     := 0;                ///***
         ELSE
				nDel	:= 2;												// formatovanie na stred
            IF x4o^.fil[i] THEN
                ii := 0;                       				// FgC - farba popredia kruznice bude cierna
             ELSE
               ii := x4o^.BgC[i];                    		// farba
            END_IF;
            IF x4o^.txt[i] THEN
               del   := 0;
               jj    := 0;
					IF x4o^.obr[i] >= 10000 THEN					// predsadi pred/za obrazok
						nNew := x4o^.obr[i] - 10000;
						IF i = 1 OR i = 3 THEN						// vlavo pred objekt
							nDel	:= 1;									// <--
							x		:= xO2^.x - xO2^.w*10/3 ;
						ELSE
							x		:= xO2^.x + xO2^.w/2 + xO2^.w/10 ;
							nDel	:= 0;									// -->
						END_IF;
					ELSE
						nNew := x4o^.obr[i];
					END_IF;
               yTx1  := INT_TO_STRING(nNew);      // cislo z obrazka sa prevedie na text
            ELSE
               del   := x4o^.obr[i];               		// bude cislo obrazka
               jj    := -1;
            END_IF;
				o	:= USINT_TO_INT(x4o^.wxy[i]);
				IF x4o^.crc[i] THEN
               IF x4o^.txt[i]  THEN
                  grp := grp * 20 / 39;
						IF x4o^.obr[i] > 99 THEN
							o := o*10/7;
						END_IF;
//               ELSIF x4o^.fil[i] = false THEN
					ELSE
                  grp := grp * 10 / 11;

               END_IF;
            END_IF;
                     _NhVal2(
                                 crc   := x4o^.crc[i],
                                 wC    := o,
                                 grd   := 2,                                  // kruh s oramovanim bez gradientu
                                 wL    := 1,                                  // hrubka kruznice
                                 fil   := x4o^.fil[i],
                                 xy    := true,                               // move to x,y
                                 x     := x,
                                 y     := y,
                                 obr   := del,                        // >0 obrazok, <=0 ignoruje, je to text
                                 wO    := grp,
                                 wT    := grp,
                                 fmt   := nDel,
                                 txt   := jj,
                                 FgT   := x4o^.FgT[i],
                                 FgC   := ii,
                                 BgC   := x4o^.BgC[i]
                              );

         END_IF;
      END_IF;
   END_FOR;
END_FUNCTION

FUNCTION _NhDayObr {HIDDEN}: INT      // vykreslit doplnujuce objektynad hlavnym objektom, dotyk a cykonanie pripadneho CMD
   VAR_INPUT
      off   : BOOL;
      day   : SINT;
   END_VAR
   CASE day OF
     0 : _NhDayObr := 140;
     1 : _NhDayObr := 142;
     2 : _NhDayObr := 144;
     3 : _NhDayObr := 146;
    10 : _NhDayObr := 148;      // vychod slnka
    11 : _NhDayObr := 147;      // zapad slnka
   END_CASE;
   IF off THEN
      _NhDayObr := _NhDayObr - 1;
   END_IF;
END_FUNCTION

FUNCTION _Nh_FRM_Read_SLIDER {HIDDEN}: BOOL
	IF yFrmName.sld > 0 THEN                                                     		// mame slider
		OffSrc := USINT_TO_UDINT(yFrmName.row) * SIZEOF(NH_ROW_O);          				// slider zacina za riadkami browsu
		OffDst := (yFrmName.siz - SIZEOF(NH_FRM_HED) - OffSrc) / SIZEOF(NH_SLD_DAT) ;	// kolko riadkov realne obsahuju zvysne data
//		OffDst := USINT_TO_UDINT(yFrmName.sld);
		memCpyPTR(	source	:= ADR(yFrmData) + offSrc ,											// adresa zaciatku slidera
						dest		:= PTR_TO_UDINT(ADR( xB^.s[0] )) ,	                     // kopiruje sa do slidera 0
						length	:= OffDst * SIZEOF(NH_SLD_DAT) );                        // pocet sliderov * velkost slidera {ak bude 0 tak sa nic nekopiruje}
	END_IF;
END_FUNCTION

FUNCTION  _NhIsObrOk {HIDDEN}: BOOL (* yTx1:=CONCAT('_',UINT_TO_STRINGF(frm,'%03u')); yTx2:=CONCAT(aSys.ADR_RAM,'FRM/',yTx1,'.FRM'); *)
	VAR_INPUT
		frm	: UINT;
	END_VAR
//	yTx0 := CONCAT('_',UINT_TO_STRINGF(frm,'%03u'));
	rb := _Nh_Log_PATH(wh:=24, frm:=7, obr:=frm); 		//yTx2:='_999", yTx1:='RAM/FRM/_999.FRM'
// 	If yFrmName.Name = yTx0 THEN
 	If yFrmName.Name = yTx2 THEN
		_NhIsObrOk := TRUE;
		RETURN;
	ELSE
		_NhIsObrOk := false;
	END_IF;
//	fH 	:= INVALID_HANDLE_VALUE;
//	yTx0 	:= CONCAT(aSys.DiskHed.Disk[4].path,'FRM/',yTx0,'.FRM');							// RAM/
//  	IF _NhFOpen(fN:=yTx0, fH:=fH) THEN
  	IF _NhFOpen(fN:=yTx1, fH:=fH) THEN
     	yFrmName.siz 	:= fS;
  		yFrmName.siz 	:= FileRead  (hFile := fH, adrBuf := PTR_TO_UDINT(ADR(mObr)), size := fS );
		_NhIsObrOk		:= yFrmName.siz = fS;
		rb					:= _NhFClose(fH:=fH);
	END_IF;
END_FUNCTION

FUNCTION _Nh_FRM_Read {HIDDEN}: BOOL
   VAR_INPUT
		ref		: BOOL;
      frm      : UINT;          // pripona suboru
      row      : USINT;
   END_VAR
   VAR_TEMP
      i        : USINT;
   END_VAR
  	If _NhIsObrOk(frm := frm) THEN
		_Nh_FRM_Read := TRUE;
		If ref THEN
			RETURN;
		END_IF;
	ELSE
		_Nh_FRM_Read := false;
		RETURN;
	END_IF;
	CASE yFrmName.wht OF
     0 :	// all file for next specific use
			;
     1 :	// browser
			offSrc := SIZEOF(NH_ROW_O) * USINT_TO_UDINT( MIN(yFrmName.row,xL^.dsh-1) ); 		// posun na konkretny riadok podla DSH
			memCpyPTR(	source	:= ADR(yFrmData) + offSrc ,                              		// z konkretneho riadka
							dest		:= PTR_TO_UDINT(ADR( xB^.r[row].o )) ,								// do aktualneho riadka
							length	:= SIZEOF(NH_ROW_O) );                                   	// velkost 10 objektov
			IF yFrmName.sld > 0 THEN                                                     		// mame slider
				OffSrc := USINT_TO_UDINT(yFrmName.row) * SIZEOF(NH_ROW_O) + USINT_TO_UDINT(xL^.dsh-1) * SIZEOF(NH_SLD_DAT);          				// slider zacina za riadkami browsu
				memCpyPTR(	source	:= ADR(yFrmData) +	OffSrc, 													// zaciatok DASH-1

								dest		:= PTR_TO_UDINT(ADR( xB^.s[row] )) ,	                     // kopiruje sa do slidera 0
								length	:= SIZEOF(NH_SLD_DAT) );                        // pocet sliderov * velkost slidera {ak bude 0 tak sa nic nekopiruje}
			END_IF;

//			_Nh_FRM_Read_SLIDER();

     2 :	// FRM
     		xRowO := ADR(yFrmData);
			FOR i := 1 TO yFrmName.row DO
				IF xB^.r[i].h.nd = 0 THEN
					xB^.r[i].h.nd 	:= USINT_TO_INT(i) ;
				END_IF;
				xB^.r[i].o		:= xRowO^;
				xRowO				:= xRowO + SIZEOF(NH_ROW_O);
         END_FOR;
			_Nh_FRM_Read_SLIDER();
     3 :	// menu
			i		:= xM^.lvl;
			memCpyPTR(	source	:= PTR_TO_UDINT(ADR(yFrmData)) ,
							dest		:= PTR_TO_UDINT(ADR(xM^.mnu[i])) ,
							length	:= SIZEOF(NH_MNU) );
     4 :	// HOME-PG - ALL
     		xRowO := ADR(yFrmData);
			FOR i := 0 TO yFrmName.row  DO
				xB^.r[i].h.nd 	:= USINT_TO_INT(i) ;
				xB^.r[i].o		:= xRowO^;
				xRowO				:= xRowO + SIZEOF(NH_ROW_O);
			END_FOR;
   END_CASE;

END_FUNCTION

FUNCTION _Nh_Get_Frm260  {HIDDEN} : BOOL					//
	VAR_INPUT
		cmd	: BOOL;
		cf		: USINT;
		nd		: INT;
		grp	: USINT;
	END_VAR
	_Nh_Get_Frm260 := _NhIsObrOk(frm:=260);
	_NhxPt (c := cf, n := nd,x:=35);
	yFrm_260.typ := xPt^.cf.typ;											   // typ vyssej casti
	yFrm_260.grp := grp;

		yFrm_260.m := 0;
		FOR i := 0 TO yFrm_260.nWsb DO
			IF yFrm_260.mWsb[i].mWsb = grp AND			// presna skupina
				( 	yFrm_260.mWsb[i].typ = yFrm_260.typ OR       // konkretny typ
					yFrm_260.mWsb[i].typ = -1)             		// plati pre vsetky typy
				THEN
				yFrm_260.m := i;
				EXIT;
			END_IF;
	  	END_FOR;
		IF cmd THEN
			pWsb^.cm.cmd	:= yFrm_260.mWsb[yFrm_260.m].pvCmd;
		ELSE
			xOh^.cf			:= yFrm_260.mWsb[yFrm_260.m].cf;
			xOh^.txt			:= yFrm_260.mWsb[yFrm_260.m].txt;
		END_IF
END_FUNCTION

VAR_GLOBAL
	_NhBrwObj 						: NH_BRW_OBJ;
//   _eRowBrw6      {HIDDEN} : NH_ROW_O ;         // pre kompatibilitu sa niekde pouziva
END_VAR

FUNCTION _NhTypObr  {HIDDEN} : BOOL
	VAR_INPUT
   	cf 		: USINT;
   	typ		: SINT;
		dev		: USINT;
		txx		: USINT;
	END_VAR
	cf 	:= LIMIT(cf ,0,_Nh_CFG);
	dev	:= LIMIT(dev,0,_Nh_CFG);
	_NhTypObr 	:= true;
//	xTypObr 		:= ADR(mObr);
  	If _NhIsObrOk(frm := 230) THEN
		_NhTypObr := TRUE;
	ELSE
		_NhTypObr := false;
		RETURN;
	END_IF;
	CASE cf OF
 		13: 	// WSB
      		typ := MAX(1,typ/2);
	END_CASE;

	txx	:= yFrm_230.obr[cf ].wht;
//	typ   := LIMIT(ABS(typ),0, 5);
  	CASE  yFrm_230.obr[cf ].obr OF
   	-5 : 	xObrWht 		:= ADR(yFrm_230.T05[ txx ,  typ ].obr );
				_NhTypObr   := yFrm_230.T05[ txx ,  typ ].fil[dev] OR yFrm_230.T05[ txx , typ ].fil[0] ;
     -10 : 	xObrWht 		:= ADR(yFrm_230.T10[ txx ,  typ ].obr );
				_NhTypObr   := yFrm_230.T10[ txx ,  typ ].fil[dev] OR yFrm_230.T10[ txx , typ ].fil[0] ;
     -15 : 	xObrWht 		:= ADR(yFrm_230.T15[ txx ,  typ ].obr );
				_NhTypObr   := yFrm_230.T15[ txx ,  typ ].fil[dev] OR yFrm_230.T15[ txx , typ ].fil[0] ;
	//			_NhTypObr   := true;	//yFrm_230.T15[ txx ,  typ ].fil[dev] OR yFrm_230.T15[ txx ,  0 ].fil[dev] ;
	ELSE	xObrWht := ADR(yFrm_230.obr[cf ]);
   END_CASE;
END_FUNCTION

FUNCTION _Nh_POI_INI_REC {HIDDEN}   : INT	    // urobi testy POI, prida nove, vymaze stare
	_Nh_POI_INI_REC := 0;
	FOR i := 1 TO _Nh_CFG DO
		IF aCfg[i].NbrPoi > 0 THEN
		   _Nh_POI_INI_REC := _Nh_POI_INI_REC + ( 11 * ( aCfg[i].rec * USINT_TO_INT(aCfg[i].NbrPoi)) );
		END_IF;
   END_FOR;
END_FUNCTION

// HET _Nh_POI_INI_NEW(cf:=xR^.h.cf.c, nd1:=xR^.h.cf.n, nd2:=xR^.h.cf.n, del:=true);

FUNCTION _Nh_POI_INI_NEW {HIDDEN} : BOOL	// skontroluje vetu POI alebo ju vytvori zo sablony pre zadane CFG a POI
											// NESMIE SA SPUSTAT NARAZ DEL A NEW !!!!
   VAR_INPUT
//		new	: BOOL;					// vsetky POI vynulovat a nanovo pridelit
		del	: BOOL;					// len vymaze POI, nic ine
      cf   	: USINT 	:= 1;
      nd1   : INT		:= 1;       // 1.rec z ROM/HET/VEN...
      nd2   : INT;               // posledne rec
		po1	: USINT 	:= 1;       // ktory den z poi[]
		po2	: USINT 	:= 11;
   END_VAR
	VAR_TEMP
		ok2			: BOOL;
		day			: USINT;
		WhtPoi		: USINT;
		RecPoiReQ	: INT;
	END_VAR
   _Nh_POI_INI_NEW := true;
	RecPoiReQ :=_Nh_POI_INI_REC();				// na zaciatku sa spocita, kolko viet je potrebne

   _Nh_FRM_Read(frm:=247);
	IF nd2 = 0 THEN
		nd2 := aCfg[cf].rec;
	END_IF;
  	day	:= po1;
   WHILE nd1 <= nd2  DO                                		// pre CF
		ok2 := true;
		IF _Nh_xPod_Map(cf:=cf, nd:=nd1, WhtPoi:=WhtPoi) THEN                // veta ROM/HET/VEN, musi sa vzdy premapovat po pridani novych viet do POI
			IF xPod^.Day = 0 OR xPod^.Day > 11 THEN
         	xPod^.Day := SYSTEM_S.COUNTER_DAYS_OF_WEEK;										// kontrola na 0-day
			END_IF;
			WHILE day <= po2 DO
				IF del OR xPod^.poi[day] < 0 OR xPod^.poi[day] > aCfg[26].rec THEN									// vymaze stare alebo neplatne (-1) POI ak existuje a prida vzdy odkaz na novu vetu POI
					IF xPod^.poi[day] > 0 AND xPod^.poi[day] <= aCfg[26].rec THEN  // veta existuje
						IF _NhxPt(ok:=1, c:=26, n:=xPod^.poi[day], x:=-124) THEN  	// najde vetu aby ju vymazal
							xPt^.ok.ok := false;                 							// len zneplatni, neprepisuje udaje
						END_IF;
					END_IF;
					xPod^.poi[day] := 0;                                  			// vynuluje cislo vety pre day
				END_IF;
				IF del  THEN                     						// len vymnazava, alebo opravuje, a nepridava
					;
				ELSIF xPod^.poi[day] = 0 THEN                      					// ak nename POI vetu, hlada sa DEL veta
					; //vyriesi sa dalej
				ELSIF _NhxPt(ok:=1, c:=26, n:=xPod^.poi[day], x:=-124) = false THEN    // nenasla sa ani DEL veta
					xPod^.poi[day] := 0;
				END_IF;
				IF del THEN              									// len vymnazava, alebo opravuje
					day 	:= day + 1;
				ELSIF xPod^.poi[day] = 0 THEN													// nebola najdena DEL veta
					ok1	:= false;
					IF aCfg[26].rec >= RecPoiReQ THEN	//_Nh_POI_INI_REC() THEN
						xPod^.poi[day] := _NhFindDel(wh:=0, cx:=26, new:=false, ok:=true); 	// ak najde vetu,oznaci ju ako OK
						IF xPod^.poi[day] > 0 THEN
							// xDel je uz namapovane a veta je OK
							xPox := xDel;
(*
						   yTx2  := CONCAT('  cf;nd;day;poi[day]: ',USINT_TO_STRINGF(cf,'%2u'),';',INT_TO_STRINGF(nd1,'%4u'),';',USINT_TO_STRINGF(day,'%2u'),';',INT_TO_STRINGF(xPod^.poi[day],'%4u')    )  ;
							yTx2  := CONCAT(yTx2,';',USINT_TO_STRINGF(WhtPoi,'%2u'),';',BOOL_TO_STRINGF(xPox^.ok.ok,'%b{on^off}'));
							_Nh1RowTxt(logRst:=1);
*)
							CASE cf OF
   	                 6 : xPox2 := ADR(yFrm_247.ini.HET);
      	             47 : xPox2 := ADR(yFrm_247.ini.VEN);
         	         ELSE  xPox2 := ADR(yFrm_247.ini.DAY);
            	      END_CASE;
							xPox2 		:= xPox2 + (SIZEOF(NH_POI) * USINT_TO_UDINT(day-1));	// zdroj=sablona
							xPox^			:= xPox2^;													// nakopiruje zo sablony
//							xPox^.ok.ok	:= true;
							day 			:= day + 1;
						ELSE
							ok1	:= true;
						END_IF;
					ELSE
						ok1	:= true;
					END_IF;
					IF ok1 THEN
						aCfg[26].new := aCfg[26].new + (11 * USINT_TO_INT( aCfg[cf].NbrPoi ));		// prida rovno 11 viet, resp kolko zostava do 11
						aCfg[26].nOk := false;                                         // neoznaci ako OK
						_Nh_Go_DbxToMem(ram := true);
						ok2 			:= false;
						RecPoiReQ 	:=_Nh_POI_INI_REC();				// len v pripade, ze by sa nenasla DEF-veta
						EXIT;
					END_IF;
				ELSE
					day := day + 1;
				END_IF;
			END_WHILE;		// day
		ELSE
			WhtPoi   := 200;												// len  aby sa posunul
		END_IF;
		IF ok2 THEN  																				// vykonali sa vsetky poi[1..11] v jednej vete CF, ide sa na dalsiu
			IF WhtPoi + 1 < aCfg[cf].NbrPoi THEN
				WhtPoi 	:= WhtPoi + 1;
			ELSE
				WhtPoi 	:= 0;
				nd1 		:= nd1 + 1;
			END_IF;
			day	:= po1;
		END_IF;
	END_WHILE;
END_FUNCTION

FUNCTION _NhFilDev  {HIDDEN} : BOOL
   VAR_INPUT
		lst	: BOOL;
		clear	: BOOL;
      wht   : USINT;
      row   : USINT;
      n     : USINT;
   END_VAR
	_NhFilDev := TRUE;
	{ $ IFDEF __NH_WEB }
	IF lst THEN
	  	IF _NhIsObrOk(frm := 236) THEN
		   CASE wht OF
   		  0 : ; // vsetky filtre vo filt
	   	  1 : xF^.dev  := yFrm_236.rgbwa;       						// ktore DEV maju HW nahradene DLs + RGBWA
   		  2 : xF^.dev  := yFrm_236.iodev[row];
	   	  3 : xF^.dev  := yFrm_236.lst[row];
	   	END_CASE;
		END_IF;
	ELSIF _NhIsObrOk(frm := 234) THEN					// vlozi do xF^.dev zoznam DEV, vyhovoujucich browsu
		IF clear OR wht = 0 THEN
			xF^.dev := yFrm_234.iov[0];					// clear dev-list
			xF^.cat := yFrm_234.iov[0];					// clear dev-list
		END_IF;
	   CASE wht OF
   	  0 : ; // vsetky filtre vo filt
	     1 : xF^.dev		:= yFrm_234.rom[row];
   	  2 : xF^.dev  	:= yFrm_234.zon[row];
   	  4 : xF^.dev  	:= yFrm_234.iov[row];
//	     5 : _NhFilDev 	:= xF^.dev.n[n];	// len frati, ci DEV je v dev-liste
	     5 : _NhFilDev 	:= yFrm_234.in[row].n[n];	// len vati, ci DEV je v dev-liste
     	  7 : xF^.dev  	:= yFrm_234.set[row];
	   END_CASE;
		RETURN;
	ELSE
		RETURN;
	END_IF;
	{ $ END_IF }
END_FUNCTION

(* ---- _Nh_WRK.st ---- *)
{ $IFDEF __NH_WRK }

VAR_GLOBAL                                            // len pre ladenie
   _NhWrk      {HIDDEN} : BOOL := true ;
   { $ IF CPU_CODE > 1999  }
   yIdx         : ARRAY[1..30]	OF NH_IDX;

	yScn			{HIDDEN} : ARRAY[1..50]  OF NH_SCN;
   ypScn 		{HIDDEN} : ARRAY[1..20]  OF NH_SVA_PAR;
	yAct			{HIDDEN} : ARRAY[1..50]  OF NH_ACT;
//	yAla			{HIDDEN} : ARRAY[1..10]  OF NH_ALA;

//		yyVaz	{HIDDEN}	: ARRAY[1.._Nh_VAZ] OF NH_VAZ_CFG ;

		yVaz1			{HIDDEN} : ARRAY[1..50]  OF NH_VAZ;
//	  	yVaz2 		{HIDDEN} : ARRAY[1..150] OF NH_VAZ;
//		yVaz3			{HIDDEN} : ARRAY[1..50]  OF NH_VAZ;
//   	yVaz4			{HIDDEN} : ARRAY[1..80]  OF NH_VAZ;

//  		yGlb			{HIDDEN} : ARRAY[1..1]   OF NH_GLB;
	   yRom			{HIDDEN} : ARRAY[1..30]	OF NH_ROM;
   	yZon			{HIDDEN} : ARRAY[1..10]	OF NH_ROM;
	   ypZon 		{HIDDEN} : ARRAY[1..20]  OF NH_ZON_PAR;
   	yRoW        {HIDDEN} : ARRAY[1..10]  OF NH_WRK_ROM;
		yZoW        {HIDDEN} : ARRAY[1.. 7]  OF NH_WRK_ROM;
		yRol			{HIDDEN} : ARRAY[1..20]  OF NH_ROL;
   	ypRol 		{HIDDEN} : ARRAY[1..100]  OF NH_ROL_PAR;       // 12
//   	yPoi			{HIDDEN} : ARRAY[1..50]  OF NH_POI;

		yTgl			{HIDDEN} : ARRAY[1..30]  OF NH_TGL;
  		ypTgl 		{HIDDEN} : ARRAY[1..120]  OF NH_WSB_PAR;

   ySvd 			{HIDDEN} : ARRAY[1..10]  OF NH_SVD;
   pSvd 			{HIDDEN} : ARRAY[1..100]  OF NH_SVD_PAR;
  	ySva 			{HIDDEN} : ARRAY[1..10]  OF NH_SVA;  //10
  	pSva 			{HIDDEN} : ARRAY[1..40]  OF NH_SVA_PAR;
   yRgb 			{HIDDEN} : ARRAY[1..10]  OF NH_RGB;
	yyRgb 			{HIDDEN} : NH_RGB;
   pRgb 			{HIDDEN} : ARRAY[1..20]  OF NH_RGB_PAR;

	yTve			{HIDDEN} : ARRAY[1..20]  OF NH_TVE;
//	yHet			{HIDDEN} : ARRAY[1..10]  OF NH_HET;  // 20
(*

 	ypHet 		{HIDDEN} : ARRAY[1..20]  OF NH_HET_PAR;       // 10

//	yHev			{HIDDEN} : ARRAY[1..5]   OF NH_HET;  // 20

	yVen 			{HIDDEN} : ARRAY[1..10]  OF NH_TVE;
*)

(*
		yLux			{HIDDEN} : ARRAY[1..5]  OF NH_LUX;
   	yTer 			{HIDDEN} : ARRAY[1..40]  OF NH_TER;
	   yTeh 			{HIDDEN} : ARRAY[1.. 5]  OF NH_TER;
   	yTek 			{HIDDEN} : ARRAY[1.. 5]  OF NH_TER;

*)
//		yRhx			{HIDDEN} : ARRAY[1..2]  OF NH_LUX;
//	yCer			{HIDDEN} : ARRAY[1..3]	 OF NH_TVE;
//	yKot			{HIDDEN} : ARRAY[1..5]	 OF NH_TVE;
//  	yTim			{HIDDEN} : ARRAY[1..10]  OF NH_TIM;
//	yKey			{HIDDEN} : ARRAY[1..3]   OF NH_KEY;

(*
	yDls			{HIDDEN} : ARRAY[1..130]   OF NH_DLS;
	pDls			{HIDDEN} : ARRAY[1..200]   OF NH_RGB_PAR;
	yDlm			{HIDDEN} : ARRAY[1..4]   OF NH_DLM;
	yDlg			{HIDDEN} : ARRAY[1..32]   OF NH_DLG;
*)

//    	yMsg			{HIDDEN} : ARRAY[1..3] OF NH_MSG;

//	  yCat			{HIDDEN} : ARRAY[1..70]	OF NH_CAT;

      yVvo 			{HIDDEN} : ARRAY[1..4]   OF NH_VVO;

   yWsb 			{HIDDEN} : ARRAY[1..30]  OF NH_WSB;
   ypWsb 		{HIDDEN} : ARRAY[1..50]  OF NH_WSB_PAR;

   yTla 			{HIDDEN} : ARRAY[1..10]  OF NH_TLA;

//   ytGl		 {HIDDEN} : ARRAY[1..10]  OF NH_TGL;
//	yPIR			{HIDDEN} : ARRAY[1..50]  OF NH_PIR;
//   ypPir 		{HIDDEN} : ARRAY[1..10]  OF NH_PIR_PAR;

//	yCox			{HIDDEN} : ARRAY[1..10]  OF NH_LUX;

//	yDor			{HIDDEN} : ARRAY[1..10]  OF NH_DOR;

//	yFav			{HIDDEN} : ARRAY[1..10]  OF NH_FAV;
//   yZas 			{HIDDEN} : ARRAY[1..15]  OF NH_SVD;
//   pZas 			{HIDDEN} : ARRAY[1..10]  OF NH_SVD_PAR;
//	yyUsr			{HIDDEN} : ARRAY[1..7]   OF NH_USR;

//	ySmw			{HIDDEN} : ARRAY[1..10]  OF NH_SMW;

//	yGat			{HIDDEN} : ARRAY[1.. 5]  OF NH_GAT;
//	yBra			{HIDDEN} : ARRAY[1.. 5]  OF NH_GAT;
//   ypGat 		{HIDDEN} : ARRAY[1..10]  OF NH_GAT_PAR;       // 13

//	ySir			{HIDDEN} : ARRAY[1.. 5]  OF NH_SVD;
//	yBlk			{HIDDEN} : ARRAY[1.. 5]  OF NH_BLK;
//	yBlx			{HIDDEN} : ARRAY[1.. 5]  OF NH_BLX;
//	yBtn			{HIDDEN} : ARRAY[1..20]  OF NH_BTN;
(*
//	yAcl			{HIDDEN} : ARRAY[1..20]  OF NH_VAZ;
*)
//	yVcf			{HIDDEN} : ARRAY[1..150]  OF NH_VAZ_VCF;
//	ySbj			{HIDDEN} : ARRAY[1..4]  OF NH_SBJ;

   { $ ELSE  }

//   	yPoi			{HIDDEN} : ARRAY[1..20]  OF NH_POI;
//	   yRom			{HIDDEN} : ARRAY[1..10]	    OF NH_ROM;
//   	yZon			{HIDDEN} : ARRAY[1..10]	  OF NH_ROM;
//    yRoW        {HIDDEN} : ARRAY[1..10]    OF NH_WRK_ROM;
   { $ END_IF  }

END_VAR

	FUNCTION	_DevDataX {HIDDEN} : BOOL
      VAR_IN_OUT
         aNh   : NH_CFG_CFG;
         dst   : USINT;
      END_VAR
      VAR_INPUT
         n    : UDINT := 10;
      END_VAR
      memsetEx(val := 0,length := n * aNh.Siz , dest := dst ); // vycisti
      IF aNh.Ram > 0 THEN
         MemcpyEx(length := Min(n, INT_TO_UDINT(aNh.Rec)) * aNh.Siz , source := void( mRam[ aNh.Ram ]), dest := dst);
      END_IF;
      _DevDataX := true;
   END_FUNCTION

   FUNCTION	_NhDataWrk {HIDDEN} : BOOL
      VAR_INPUT
         Yes  : BOOL := true ;
      END_VAR
      IF Yes = false THEN
         RETURN;
      END_IF;
		_NhDataWrk :=  TRUE;
      { $ IF CPU_CODE > 1999  }
         { $IFDEF yGlb }
            _DevDataX(aNh := VOID(aCfg[25]), dst := VOID(yGlb), n :=1);
         { $END_IF }
         { $IFDEF yRom }
            _DevDataX(aNh := VOID(aCfg[ 1]), dst := VOID(yrom), n :=30);
         { $END_IF }
         { $IFDEF yPoi }
            _DevDataX(aNh := VOID(aCfg[26]), dst := VOID(yPoi), n := 50);
         { $END_IF }
      { $ ELSE  }
         { $IFDEF yRom }
            _DevDataX(aNh := VOID(aCfg[ 1]), dst := VOID(yrom), n :=10);
         { $END_IF }
         { $IFDEF yPoi }
            _DevDataX(aNh := VOID(aCfg[26]), dst := VOID(yPoi), n := 20);
         { $END_IF }
      { $ END_IF  }

      { $IFDEF yMsg }
      _DevDataX(aNh := VOID(aCfg[46]), dst := VOID(yMsg), n :=3);
      { $END_IF }

      { $IFDEF ycat }
      _DevDataX(aNh := VOID(aCfg[ 2]), dst := VOID(yCat), n :=70);
      { $END_IF }
      { $IFDEF yZon }
      _DevDataX(aNh := VOID(aCfg[ 3]), dst := VOID(yZon), n :=10);
      { $END_IF }
      { $IFDEF ypZon }
      _DevDataX(aNh := VOID(aPar[5]), dst := VOID(ypZon), n :=20);
      { $END_IF }
      { $IFDEF yHet }
      _DevDataX(aNh := VOID(aCfg[ 6]), dst := VOID(yHet));
      { $END_IF }
      { $IFDEF yHev }
      _DevDataX(aNh := VOID(aCfg[47]), dst := VOID(yHev), n:=5);
      { $END_IF }
      { $IFDEF yKot }
      _DevDataX(aNh := VOID(aCfg[ 7]), dst := VOID(yKot), n:=5);
      { $END_IF }
      { $IFDEF ytve }
      _DevDataX(aNh := VOID(aCfg[ 8]), dst := VOID(yTve), n:=20);
      { $END_IF }
      { $IFDEF ycer }
      _DevDataX(aNh := VOID(aCfg[ 9]), dst := VOID(yCer), n := 3);
      { $END_IF }
      { $IFDEF ysvd }
      _DevDataX(aNh := VOID(aCfg[10]), dst := VOID(ySvd));
      { $END_IF }
      { $IFDEF ySva }
      _DevDataX(aNh := VOID(aCfg[11]), dst := VOID(ySva));
      { $END_IF }
      { $IFDEF yVvo }
      _DevDataX(aNh := VOID(aCfg[49]), dst := VOID(yVvo), n :=4);
      { $END_IF }
      { $IFDEF yRgb }
      _DevDataX(aNh := VOID(aCfg[12]), dst := VOID(yRgb));
      { $END_IF }
      { $IFDEF ywsb }
      _DevDataX(aNh := VOID(aCfg[13]), dst := VOID(yWsb), n :=30);
      { $END_IF }
      { $IFDEF ytla }
      _DevDataX(aNh := VOID(aCfg[14]), dst := VOID(yTla));
      { $END_IF }
      { $IFDEF ypir }
      _DevDataX(aNh := VOID(aCfg[15]), dst := VOID(yPir), n :=50);
      { $END_IF }
      { $IFDEF yter }
      _DevDataX(aNh := VOID(aCfg[16]), dst := VOID(yTer), n :=40);
      { $END_IF }
      { $IFDEF yteh }
      _DevDataX(aNh := VOID(aCfg[17]), dst := VOID(yTeh), n := 5);
      { $END_IF }
      { $IFDEF ytek }
      _DevDataX(aNh := VOID(aCfg[18]), dst := VOID(yTek), n := 5);
      { $END_IF }
      { $IFDEF ylux }
      _DevDataX(aNh := VOID(aCfg[19]), dst := VOID(yLux), n := 5);
      { $END_IF }
      { $IFDEF yRhx }
      _DevDataX(aNh := VOID(aCfg[51]), dst := VOID(yRhx), n := 2);
      { $END_IF }
      { $IFDEF yfav }
      _DevDataX(aNh := VOID(aCfg[20]), dst := VOID(yFav));
      { $END_IF }
      { $IFDEF yzas }
      _DevDataX(aNh := VOID(aCfg[21]), dst := VOID(yZas), n:=15);
      { $END_IF }
      { $IFDEF yDor }
      _DevDataX(aNh := VOID(aCfg[33]), dst := VOID(yDor));
      { $END_IF }
      { $IFDEF yyUsr }
      _DevDataX(aNh := VOID(aCfg[22]), dst := VOID(yyUsr), n:=7);
      { $END_IF }
      { $IFDEF yven }
      _DevDataX(aNh := VOID(aCfg[23]), dst := VOID(yVen));
      { $END_IF }
      { $IFDEF yKey }
      _DevDataX(aNh := VOID(aCfg[24]), dst := VOID(yKey), n := 3);
      { $END_IF }
      { $IFDEF ysmw }
      _DevDataX(aNh := VOID(aCfg[45]), dst := VOID(ySmw));
      { $END_IF }
      { $IFDEF yRol }
      _DevDataX(aNh := VOID(aCfg[31]), dst := VOID(yRol), n:=20);                    //ROL
      { $END_IF }
      { $IFDEF yBra }
      _DevDataX(aNh := VOID(aCfg[37]), dst := VOID(yBra), n := 5);            //BRA - stara
      { $END_IF }
      { $IFDEF yGat }
      _DevDataX(aNh := VOID(aCfg[37]), dst := VOID(yGat), n := 5);            //BRA
      { $END_IF }
      { $IFDEF ySir }
      _DevDataX(aNh := VOID(aCfg[32]), dst := VOID(ySir), n := 5);            //SIR
      { $END_IF }
      { $IFDEF yBlk }
      _DevDataX(aNh := VOID(aCfg[35]), dst := VOID(yBlk), n := 5);            //BLK
      { $END_IF }
      { $IFDEF yBlx }
      _DevDataX(aNh := VOID(aCfg[36]), dst := VOID(yBlX), n := 5);            //BLK
      { $END_IF }
      { $IFDEF yTgl }
      _DevDataX(aNh := VOID(aCfg[40]), dst := VOID(yTgl), n :=30);
      { $END_IF }
      { $IFDEF yBtn }
      _DevDataX(aNh := VOID(aCfg[41]), dst := VOID(yBtn), n := 20);
      { $END_IF }
      { $IFDEF yDlm }
      _DevDataX(aNh := VOID(aCfg[42]), dst := VOID(yDlm), n := 4);
      { $END_IF }
      { $IFDEF yDls }
      _DevDataX(aNh := VOID(aCfg[43]), dst := VOID(yDls), n := 130);
      { $END_IF }
      { $IFDEF yDlg }
      _DevDataX(aNh := VOID(aCfg[44]), dst := VOID(yDlg), n := 32);
      { $END_IF }
      { $IFDEF yTim }
      _DevDataX(aNh := VOID(aCfg[50]), dst := VOID(yTim), n := 10);
      { $END_IF }
      { $IFDEF yScn }
      _DevDataX(aNh := VOID(aCfg[ 4]), dst := VOID(yScn), n := 50);
      { $END_IF }
      { $IFDEF yact }
      _DevDataX(aNh := VOID(aCfg[ 5]), dst := VOID(yAct), n:= 50);
      { $END_IF }
      { $IFDEF yAla }
      _DevDataX(aNh := VOID(aCfg[48]), dst := VOID(yAla));
      { $END_IF }
      { $IFDEF yVaz1 }
      _DevDataX(aNh := VOID(aVaz[ 1]), dst := VOID(yVaz1), n := 50);
      { $END_IF }
      { $IFDEF yVaz2 }
      _DevDataX(aNh := VOID(aVaz[ 2]), dst := VOID(yVaz2), n :=150);
      { $END_IF }
      { $IFDEF yVaz3 }
      _DevDataX(aNh := VOID(aVaz[ 3]), dst := VOID(yVaz3), n := 50);
      { $END_IF }
      { $IFDEF yVaz4 }
      _DevDataX(aNh := VOID(aVaz[ 4]), dst := VOID(yVaz4), n :=80);
      { $END_IF }

(*
      { $IFDEF yAcl }
      _DevDataX(aNh := VOID(aVaz[ 5]), dst := VOID(yAcl), n := 20);
      { $END_IF }
*)

      { $IFDEF pSvd }
       _DevDataX(aNh := VOID(aPar[1]), dst := VOID(pSvd), n := 100);
      { $END_IF }
      { $IFDEF pSva }
      _DevDataX(aNh := VOID(aPar[2]), dst := VOID(pSva), n := 40);
      { $END_IF }
      { $IFDEF pRgb }
      _DevDataX(aNh := VOID(aPar[3]), dst := VOID(pRgb), n:=20);
      { $END_IF }
      { $IFDEF ypWsb }
      _DevDataX(aNh := VOID(aPar[4]), dst := VOID(ypWsb), n := 50);
      { $END_IF }
      { $IFDEF ypTgl }
      _DevDataX(aNh := VOID(aPar[15]), dst := VOID(ypTgl), n := 120);
      { $END_IF }
      { $IFDEF pTla }
      _DevDataX(aNh := VOID(aPar[5]), dst := VOID(ypTla), n:=20);
      { $END_IF }
      { $IFDEF pZas }
      _DevDataX(aNh := VOID(aPar[6]), dst := VOID(pZas));
      { $END_IF }
      { $IFDEF ypPir }
      _DevDataX(aNh := VOID(aPar[7]), dst := VOID(ypPir));
      { $END_IF }
      { $IFDEF ypHEt }
      _DevDataX(aNh := VOID(aPar[9]), dst := VOID(ypHet), n := 20);
      { $END_IF }
      { $IFDEF ypScn }
      _DevDataX(aNh := VOID(aPar[10]), dst := VOID(ypScn), n := 20);
      { $END_IF }
      { $IFDEF ypRol }
      _DevDataX(aNh := VOID(aPar[12]), dst := VOID(ypRol), n:=100);
      { $END_IF }
      { $IFDEF ypGat }
      _DevDataX(aNh := VOID(aPar[13]), dst := VOID(ypGat));
      { $END_IF }
      { $IFDEF yCox }
      _DevDataX(aNh := VOID(aCfg[41]), dst := VOID(yCox), n :=10);
      { $END_IF }
      { $IFDEF pDls }
      _DevDataX(aNh := VOID(aPar[16]), dst := VOID(pDLs), n := 200);
      { $END_IF }

// WRK
      { $IFDEF yCaW }
//         memset(val := 0, length := aSys.sCaW, dest := VOID( mRam[aSys.aCaW1] ));
         MemcpyEx(length :=  aSys.sCaW  , source := void( mRam[aSys.aCaW1] ), dest := VOID(yCaW));
      { $END_IF }
      { $IFDEF yRoW }
         MemcpyEx(length :=  MIN(10,aSys.sRoW/SIZEOF(NH_WRK_ROM))  , source := void( mRam[aSys.aRoW1] ), dest := VOID(yRoW));
      { $END_IF }
      { $IFDEF yZoW }
         MemcpyEx(length :=  MIN( 7,aSys.sRoW/SIZEOF(NH_WRK_ROM))  , source := void( mRam[aSys.aZoW1] ), dest := VOID(yZoW));
      { $END_IF }

      { $IFDEF yIdx }
         memset(val := 0, length := 30 * SIZEOF(NH_IDX), dest := VOID(yIdx));
         MemcpyEx(length :=  MIN(30,USINT_TO_UDINT(aWeb.M[1].ixb[0].idx + aWeb.M[1].ixb[1].idx)) * SIZEOF(NH_IDX)  , source := void( mRam[aSys.vIx1] ), dest := VOID(yIdx));
      { $END_IF }

   END_FUNCTION

{ $ ELSE }
   VAR_GLOBAL                                            // len pre ladenie
      _NhWrk      {HIDDEN} : BOOL := false;
   END_VAR
{ $END_IF }
